METHOD PROTECTED DriveHomeAbsSwitch : BOOL
VAR_INPUT
	Execute: BOOL;
END_VAR

VAR_INST
	
	HomeSwState: INT; 
END_VAR
VAR
	
END_VAR


IF HomeRefTrig.EDGEPOS(Execute) THEN
	HomeSwState := 1;
	DriveHomeAbsSwitch := FALSE;
END_IF


IF HomeRefTrig.EDGENEG(Execute) THEN
	
	HomeSwState := 0;
END_IF



CASE HomeSwState OF
	0:
		DriveHomeAbsSwitch := FALSE;
	1:

		IF AxisCtrlPtr^.Input.Parameter.HomeOptions.stBasic.StartDirection = eHomeModeOption.ePOSITIVE THEN
		//Sensor positive
			IF AxisCtrlPtr^.Input.Parameter.HomeOptions.stAbsSwitch.SensorEdgeSignal = eHomeModeOption.ePOSITIVE THEN
				Homing_Ctrl_Params.HomingMethod := DINT_TO_SINT(eHomingMethods.HomeAbs);
			ELSE
				Homing_Ctrl_Params.HomingMethod := DINT_TO_SINT(eHomingMethods.ForwardOnNegSw);
			END_IF
		ELSE//Direction negative
			
			IF AxisCtrlPtr^.Input.Parameter.HomeOptions.stAbsSwitch.SensorEdgeSignal = eHomeModeOption.ePOSITIVE THEN
				Homing_Ctrl_Params.HomingMethod := DINT_TO_SINT(eHomingMethods.ReverseOnPosSw);
			ELSE
				Homing_Ctrl_Params.HomingMethod := DINT_TO_SINT(eHomingMethods.ReverseOnNegSw);
			END_IF
				
		END_IF
		

		HomeSwState := 2;
		Meth_Homing(FALSE);
	2:
		IF Meth_Homing(TRUE) THEN
		  Meth_Homing(FALSE);		  
		  HomeSwState := 3;
		END_IF
		
	3:
				//homin direct
		(*IF HomeDirect(TRUE) THEN*)   		 
			Meth_CoEChangOperationMode(FALSE,eCaOpDriveModeOfOperation.CyclicSyncMode);
			
			DriveHomeAbsSwitch := TRUE;
		//END_IF	
		
		
END_CASE
END_METHOD

METHOD DriveHomeLagError : BOOL
VAR_INPUT
	Execute: BOOL;
END_VAR

VAR_INST
//	State:INT;	
//	HomeTrig: Trigger;
//	Reset:BOOL;	
//	Delay:	TON;	
	HomeLagErrState: INT; 	
	LagErrorPrevState : INT;
	
END_VAR
VAR
	
END_VAR


IF HomeRefTrig.EDGEPOS(Execute) THEN
	HomeLagErrState := 1;
	DriveHomeLagError := FALSE;
END_IF


IF HomeRefTrig.EDGENEG(Execute) THEN
	
	HomeLagErrState := 0;
END_IF



CASE HomeLagErrState OF
	0:
	//
	
	//CoEDrive_Ctrl_Adr.MaxCurrent.Index
	1:
	// set min torque
		FB_EcCoeSdoWrite.bExecute := FALSE;
		
		HomeLagErrState := HomeLagErrState + 1;
	2:
		
			FB_EcCoeSdoWrite.sNetId		:= strEcNetId;
			FB_EcCoeSdoWrite.nSlaveAddr	:= io_EtherCatAddr;
			FB_EcCoeSdoWrite.nIndex		:= CoEDrive_Ctrl_Adr.MaxCurrent.Index; 
			FB_EcCoeSdoWrite.nSubIndex	:= CoEDrive_Ctrl_Adr.MaxCurrent.SunIndex; 
			FB_EcCoeSdoWrite.pSrcBuf	:= ADR(AxisCtrlPtr^.Input.Parameter.HomeOptions.stLagErr.BlockSearchMaxCurrent);
			FB_EcCoeSdoWrite.cbBufLen	:= SIZEOF(AxisCtrlPtr^.Input.Parameter.HomeOptions.stLagErr.BlockSearchMaxCurrent);
			FB_EcCoeSdoWrite.tTimeout	:= T#10S;
	
			FB_EcCoeSdoWrite.bExecute := TRUE;
			
			HomeLagErrState := HomeLagErrState + 1;
	3:
			
	
			IF NOT FB_EcCoeSdoWrite.bBusy THEN	
				IF NOT FB_EcCoeSdoWrite.bError THEN
					FB_EcCoeSdoWrite.bExecute		:= FALSE;
					HomeLagErrState :=  HomeLagErrState + 1;
				ELSE
					HomeLagErrState := 20;//error	
				END_IF	
			END_IF
			
	4:
		
			FB_EcCoeSdoWrite.sNetId		:= strEcNetId;
			FB_EcCoeSdoWrite.nSlaveAddr	:= io_EtherCatAddr;
			FB_EcCoeSdoWrite.nIndex		:= CoEDrive_Ctrl_Adr.MaxCurrent.Index; 
			FB_EcCoeSdoWrite.nSubIndex	:= CoEDrive_Ctrl_Adr.MaxCurrent.SunIndex; 
			FB_EcCoeSdoWrite.pSrcBuf	:= ADR(AxisCtrlPtr^.Input.Parameter.HomeOptions.stLagErr.BlockSearchRatedCurrent);
			FB_EcCoeSdoWrite.cbBufLen	:= SIZEOF(AxisCtrlPtr^.Input.Parameter.HomeOptions.stLagErr.BlockSearchRatedCurrent);
			FB_EcCoeSdoWrite.tTimeout	:= T#10S;
	
			FB_EcCoeSdoWrite.bExecute := TRUE;
			
			HomeLagErrState := HomeLagErrState + 1;
	5:
			
	
			IF NOT FB_EcCoeSdoWrite.bBusy THEN	
				IF NOT FB_EcCoeSdoWrite.bError THEN
					FB_EcCoeSdoWrite.bExecute		:= FALSE;
					HomeLagErrState :=  HomeLagErrState + 1;
				ELSE
					HomeLagErrState := 22;//error	
				END_IF	
			END_IF
			
			
	6:
		
			FB_EcCoeSdoWrite.sNetId		:= strEcNetId;
			FB_EcCoeSdoWrite.nSlaveAddr	:= io_EtherCatAddr;
			FB_EcCoeSdoWrite.nIndex		:= CoEDrive_Ctrl_Adr.PositionErrorWin.Index; 
			FB_EcCoeSdoWrite.nSubIndex	:= CoEDrive_Ctrl_Adr.PositionErrorWin.SunIndex; 
			FB_EcCoeSdoWrite.pSrcBuf	:= ADR(AxisCtrlPtr^.Input.Parameter.HomeOptions.stLagErr.BlockSearchPositionWindow);
			FB_EcCoeSdoWrite.cbBufLen	:= SIZEOF(AxisCtrlPtr^.Input.Parameter.HomeOptions.stLagErr.BlockSearchPositionWindow);
			FB_EcCoeSdoWrite.tTimeout	:= T#10S;
	
			FB_EcCoeSdoWrite.bExecute := TRUE;
			
			HomeLagErrState := HomeLagErrState + 1;
	7:
			
	
			IF NOT FB_EcCoeSdoWrite.bBusy THEN	
				IF NOT FB_EcCoeSdoWrite.bError THEN
					FB_EcCoeSdoWrite.bExecute		:= FALSE;
					HomeLagErrState :=  HomeLagErrState + 1;
				ELSE
					HomeLagErrState := 20;//error	
				END_IF	
			END_IF		
			
			
	8:	
		IF WriteNC_AxisBoolParam(MC_AxisParameter:=MC_AxisParameter.EnablePosLagMonitoring,ParamValue:=FALSE) THEN
				HomeLagErrState := HomeLagErrState + 1;
			END_IF		
		
	
	9:
	

		IF AxisCtrlPtr^.Input.Parameter.HomeOptions.stBasic.StartDirection = eHomeModeOption.ePOSITIVE THEN
		//Sensor positive
 				Homing_Ctrl_Params.HomingMethod := DINT_TO_SINT(eHomingMethods.HarsrStopPosDir);
			ELSE
				Homing_Ctrl_Params.HomingMethod := DINT_TO_SINT(eHomingMethods.HarsrStopNegDir);			
		END_IF
		

		HomeLagErrState :=  HomeLagErrState + 1;
		Meth_Homing(FALSE);
	10:
		IF Meth_Homing(TRUE) THEN
		  Meth_Homing(FALSE);		
 		  HomeLagErrState :=  HomeLagErrState + 1;
		  AxisCtrlPtr^.Input.Command.Power := FALSE;
		END_IF
	11:
			FB_EcCoeSdoWrite.sNetId		:= strEcNetId;
			FB_EcCoeSdoWrite.nSlaveAddr	:= io_EtherCatAddr;
			FB_EcCoeSdoWrite.nIndex		:= CoEDrive_Ctrl_Adr.MaxCurrent.Index; 
			FB_EcCoeSdoWrite.nSubIndex	:= CoEDrive_Ctrl_Adr.MaxCurrent.SunIndex; 
			FB_EcCoeSdoWrite.pSrcBuf	:= ADR(AxisCtrlPtr^.Input.Parameter.HomeOptions.stLagErr.BlockSearchMaxCurrent);
			FB_EcCoeSdoWrite.cbBufLen	:= SIZEOF(AxisCtrlPtr^.Input.Parameter.HomeOptions.stLagErr.BlockSearchMaxCurrent);
			FB_EcCoeSdoWrite.tTimeout	:= T#10S;
	
			FB_EcCoeSdoWrite.bExecute := TRUE;
			
			HomeLagErrState := HomeLagErrState + 1;	
		
	12:
			IF NOT FB_EcCoeSdoWrite.bBusy THEN	
				IF NOT FB_EcCoeSdoWrite.bError THEN
					FB_EcCoeSdoWrite.bExecute		:= FALSE;
					HomeLagErrState :=  HomeLagErrState + 1;
				ELSE
					HomeLagErrState := 20;//error	
				END_IF	
			END_IF	
			
	13:
			FB_EcCoeSdoWrite.sNetId		:= strEcNetId;
			FB_EcCoeSdoWrite.nSlaveAddr	:= io_EtherCatAddr;
			FB_EcCoeSdoWrite.nIndex		:= CoEDrive_Ctrl_Adr.PositionErrorWin.Index; 
			FB_EcCoeSdoWrite.nSubIndex	:= CoEDrive_Ctrl_Adr.PositionErrorWin.SunIndex; 
			FB_EcCoeSdoWrite.pSrcBuf	:= ADR(AxisCtrlPtr^.Input.Parameter.HomeOptions.stLagErr.BlockExitPositionWindow);
			FB_EcCoeSdoWrite.cbBufLen	:= SIZEOF(AxisCtrlPtr^.Input.Parameter.HomeOptions.stLagErr.BlockExitPositionWindow);;
			FB_EcCoeSdoWrite.tTimeout	:= T#10S;
	
			FB_EcCoeSdoWrite.bExecute := TRUE;
			
			HomeLagErrState := HomeLagErrState + 1;	
		
	14:
			IF NOT FB_EcCoeSdoWrite.bBusy THEN	
				IF NOT FB_EcCoeSdoWrite.bError THEN
					FB_EcCoeSdoWrite.bExecute		:= FALSE;
					HomeLagErrState :=  HomeLagErrState + 1;
				ELSE
					HomeLagErrState := 20;//error	
				END_IF	
			END_IF	

	15:
		
			FB_EcCoeSdoWrite.sNetId		:= strEcNetId;
			FB_EcCoeSdoWrite.nSlaveAddr	:= io_EtherCatAddr;
			FB_EcCoeSdoWrite.nIndex		:= CoEDrive_Ctrl_Adr.MaxCurrent.Index; 
			FB_EcCoeSdoWrite.nSubIndex	:= CoEDrive_Ctrl_Adr.MaxCurrent.SunIndex; 
			FB_EcCoeSdoWrite.pSrcBuf	:= ADR(AxisCtrlPtr^.Input.Parameter.HomeOptions.stLagErr.BlockExitRatedCurrent);
			FB_EcCoeSdoWrite.cbBufLen	:= SIZEOF(AxisCtrlPtr^.Input.Parameter.HomeOptions.stLagErr.BlockExitRatedCurrent);
			FB_EcCoeSdoWrite.tTimeout	:= T#10S;
	
			FB_EcCoeSdoWrite.bExecute := TRUE;
			
			HomeLagErrState := HomeLagErrState + 1;
	16:
			
	
			IF NOT FB_EcCoeSdoWrite.bBusy THEN	
				IF NOT FB_EcCoeSdoWrite.bError THEN
					FB_EcCoeSdoWrite.bExecute		:= FALSE;
					HomeLagErrState :=  HomeLagErrState + 1;
				ELSE
					HomeLagErrState := 22;//error	
				END_IF	
			END_IF

		
	17:	
 		AxisCtrlPtr^.Input.Command.Power := TRUE;
		DriveHomeLagError:= TRUE;
	
		
END_CASE

	IF LagErrorPrevState <> HomeLagErrState THEN
		fnLogMsg(ADR(LogMsg_0),LOG_INFO,'Coe Basic Drive Lag Err step %d',HomeLagErrState,0,0);
		LagErrorPrevState := HomeLagErrState;
	END_IF
END_METHOD

METHOD PROTECTED DriveHomeRefPulse : BOOL
VAR_INPUT
	Execute: BOOL;
END_VAR

VAR_INST
	 
	RefState: INT; 
	PrevRefState : INT;
END_VAR
VAR
	
END_VAR


IF HomeRefTrig.EDGEPOS(Execute) THEN
	RefState := 1;
	DriveHomeRefPulse := FALSE;
END_IF


IF HomeRefTrig.EDGENEG(Execute) THEN
	
	RefState := 0;
END_IF



CASE RefState OF
	0:
		DriveHomeRefPulse := FALSE;
	1:
 
		IF AxisCtrlPtr^.Input.Parameter.HomeOptions.stBasic.StartDirection = eHomeModeOption.ePOSITIVE THEN
			Homing_Ctrl_Params.HomingMethod := DINT_TO_SINT(eHomingMethods.IndexPulsePosDir);
		ELSE
			Homing_Ctrl_Params.HomingMethod := DINT_TO_SINT(eHomingMethods.IndexPulseNegDir);
		END_IF	
		RefState := RefState  +1 ;
		Meth_Homing(FALSE);
	2:
		IF Meth_Homing(TRUE) THEN
		  Meth_Homing(FALSE);
		  RefState := RefState  +1 ;
		  DriveHomeRefPulse := TRUE;
		END_IF
	3:
				//homin direct
	//	IF HomeDirect(TRUE) THEN   		 
			Meth_CoEChangOperationMode(FALSE,eCaOpDriveModeOfOperation.CyclicSyncMode);
			RefState := RefState  +1 ;
	//	END_IF
	
	4: 	
	   	  DriveHomeRefPulse := TRUE;
		
		
		
END_CASE


	IF PrevRefState <> RefState THEN
		fnLogMsg(ADR(LogMsg_0),LOG_INFO,'Coe Basic Home Ref Pulse step %d',RefState,0,0);
		PrevRefState := RefState;
	END_IF
END_METHOD

METHOD DriveUnitsTorqueToRealValue : LREAL
VAR_INPUT
	
	Torque: LREAL;	

END_VAR
DriveUnitsTorqueToRealValue := Torque;
END_METHOD

METHOD EcCoeSdoRead : BOOL
VAR_INPUT
	Execute: 	BOOL;
END_VAR

VAR_INST
	CoReaderrorTrig: 		Trigger ;	
	
END_VAR

IF CoReaderrorTrig.EDGEPOS(Execute) THEN
	EcCoeSdoRead:= FALSE;
	StateCoeSdoRead	:= 1;		
END_IF

IF CoReaderrorTrig.EDGENEG(Execute) THEN
	
	CoeSdoRW.Output.Read.Done 	:= FALSE;
	FB_EcCoeSdoRead_0.bExecute 	:= FALSE;
	StateCoeSdoRead		:= 0;	
	EcCoeSdoRead		:= FALSE;
	
END_IF


CASE StateCoeSdoRead OF
	
	0:
		// Wait	
	1:
		FB_EcCoeSdoRead_0.sNetId		:= F_CreateAmsNetId(AxisCtrlPtr^.Input.Parameter.ecNetIdArr); 
		FB_EcCoeSdoRead_0.nSlaveAddr	:= io_EtherCatAddr;
		FB_EcCoeSdoRead_0.nSubIndex		:= CoeSdoRW.Input.Read.nSubIndex;
		FB_EcCoeSdoRead_0.nIndex		:= CoeSdoRW.Input.Read.nIndex; 
		FB_EcCoeSdoRead_0.pDstBuf		:= CoeSdoRW.Input.Read.pDstBuf; 
		FB_EcCoeSdoRead_0.cbBufLen		:= CoeSdoRW.Input.Read.cbBufLen; 
		FB_EcCoeSdoRead_0.tTimeout		:= CoeSdoRW.Input.Read.tTimeout; 
		StateCoeSdoRead	:= 2;
		FB_EcCoeSdoRead_0.bExecute		:= FALSE;
		
	2:	

		FB_EcCoeSdoRead_0.bExecute		:= TRUE;	
		IF (FB_EcCoeSdoRead_0.bBusy = TRUE) THEN
			StateCoeSdoRead	:= 3;	
		END_IF

	3:	
		IF (FB_EcCoeSdoRead_0.bBusy = FALSE) THEN
			
			CoeSdoRW.Output.Read.Done	:= TRUE;
			EcCoeSdoRead	:= TRUE;
			StateCoeSdoRead	:= 4;	
		END_IF
	
	4:	
		FB_EcCoeSdoRead_0.bExecute	:= FALSE;
		EcCoeSdoRead	:= TRUE;
	
		
END_CASE

FB_EcCoeSdoRead_0();

(* check if error occured *)
IF errorTrig.EDGEPOS(FB_EcCoeSdoRead_0.bError) THEN
	
	// Add FB Error to ErrorHandler	
	AddNCError(FB_EcCoeSdoRead_0.nErrId,'NC Error FB_EcCoeSdoRead_0 ErrorID: ');
	
	EcCoeSdoRead :=  FALSE ;
	FB_EcCoeSdoRead_0.bExecute := FALSE;
END_IF

CoeSdoRW.Output.Read.Busy	:= FB_EcCoeSdoRead_0.bBusy;
END_METHOD

METHOD EcCoeSdoWrite : BOOL
VAR_INPUT
	Execute: 	BOOL;
END_VAR

VAR_INST
	CanOpWriteErrorTrig: 		Trigger ;	
	
END_VAR
VAR_OUTPUT	
	Error: 	BOOL;
END_VAR

IF CanOpWriteErrorTrig.EDGEPOS(Execute) THEN
	EcCoeSdoWrite		:= FALSE;
	StateCoeSdoWrite	:= 1;		
	Error 				:= FALSE;
END_IF

IF CanOpWriteErrorTrig.EDGENEG(Execute) THEN
	
	CoeSdoRW.Output.Write.Done 	:= FALSE;
	FB_EcCoeSdoWrite_0.bExecute := FALSE;
	StateCoeSdoWrite	:= 0;	
	EcCoeSdoWrite		:= FALSE;
	
END_IF


CASE StateCoeSdoWrite OF
	
	0:
		// Wait	
	1:										   
		FB_EcCoeSdoWrite_0.sNetId		:= F_CreateAmsNetId(AxisCtrlPtr^.Input.Parameter.ecNetIdArr); 
		FB_EcCoeSdoWrite_0.nSlaveAddr	:= AxisCtrlPtr^.Input.Parameter.Drive.EtherCatAddr;
		FB_EcCoeSdoWrite_0.nSubIndex	:= CoeSdoRW.Input.Write.nSubIndex;
		FB_EcCoeSdoWrite_0.nIndex		:= CoeSdoRW.Input.Write.nIndex; 
		FB_EcCoeSdoWrite_0.pSrcBuf		:= CoeSdoRW.Input.Write.pSrcBuf; 
		FB_EcCoeSdoWrite_0.cbBufLen		:= CoeSdoRW.Input.Write.cbBufLen; 
		FB_EcCoeSdoWrite_0.tTimeout		:= CoeSdoRW.Input.Write.tTimeout; 
		StateCoeSdoWrite	:= 2;	
	2:	

		FB_EcCoeSdoWrite_0.bExecute		:= TRUE;	
		IF (FB_EcCoeSdoWrite_0.bBusy = TRUE) THEN
			StateCoeSdoWrite	:= 3;	
		END_IF

	3:	
		IF (FB_EcCoeSdoWrite_0.bBusy = FALSE) THEN
			FB_EcCoeSdoWrite_0.bExecute		:= FALSE;
			CoeSdoRW.Output.Write.Done		:= TRUE;
			EcCoeSdoWrite		:= TRUE;
			StateCoeSdoWrite	:= 4;	
		ELSIF FB_EcCoeSdoWrite_0.bError THEN
			Error := TRUE;
		END_IF
	4:
		EcCoeSdoWrite		:= TRUE;
	
	
END_CASE

FB_EcCoeSdoWrite_0();

(* check if error occured *)
IF errorTrig.EDGEPOS(FB_EcCoeSdoWrite_0.bError) THEN
	
	// Add FB Error to ErrorHandler	
	AddNCError(FB_EcCoeSdoWrite_0.nErrId,'NC Error FB_EcCoeSdoWrite_0 ErrorID: ');
	
	EcCoeSdoWrite :=  FALSE ;
	FB_EcCoeSdoWrite_0.bExecute := FALSE;
END_IF

CoeSdoRW.Output.Write.Busy	:= FB_EcCoeSdoWrite_0.bBusy;
END_METHOD

METHOD GetCanOpenAdr : BOOL
VAR_INPUT
END_VAR


VAR
	
	SpeedSwSubIndex: INT;
END_VAR
	
	CoEDrive_Ctrl_Adr.OperationMode.Index 	   := 16#6060;
	CoEDrive_Ctrl_Adr.OperationMode.SunIndex   := 0;
	CoEDrive_Ctrl_Adr.OperationMode.Size	   := 1;

	CoEDrive_Ctrl_Adr.ControlWord.Index   	 := 16#6040;	
	CoEDrive_Ctrl_Adr.ControlWord.SunIndex   := 0;
	CoEDrive_Ctrl_Adr.ControlWord.Size       := 2;
	
	
	CoEDrive_Ctrl_Adr.HomingMethod.Index  := 16#6098;
	CoEDrive_Ctrl_Adr.HomingMethod.SunIndex  := 0;
	CoEDrive_Ctrl_Adr.HomingMethod.Size      := 1;
	
	
	CoEDrive_Ctrl_Adr.HomingSWSpeed.Index     := 16#6099;		
	CoEDrive_Ctrl_Adr.HomingSWSpeed.SunIndex  := 1;
	CoEDrive_Ctrl_Adr.HomingSWSpeed.Size      := 4;
	
	
	CoEDrive_Ctrl_Adr.HomingTrSpeed.Index    := 16#6099;
	CoEDrive_Ctrl_Adr.HomingTrSpeed.SunIndex := 2;
	CoEDrive_Ctrl_Adr.HomingTrSpeed.Size     := 4;
	
	
	
	CoEDrive_Ctrl_Adr.HomingAcc.Index     	 := 16#609A;
	CoEDrive_Ctrl_Adr.HomingAcc.SunIndex  	 := 0;
	CoEDrive_Ctrl_Adr.HomingAcc.Size      := 4;
	
	CoEDrive_Ctrl_Adr.HomeOffset.Index    	 := 16#607C;
	CoEDrive_Ctrl_Adr.HomeOffset.SunIndex  	 := 0;
	CoEDrive_Ctrl_Adr.HomeOffset.Size      := 4;

	
	CoEDrive_Ctrl_Adr.StatusWord.Index     := 16#6041;
	CoEDrive_Ctrl_Adr.StatusWord.SunIndex  := 0;
	CoEDrive_Ctrl_Adr.StatusWord.Size      := 2;
	
	CoEDrive_Ctrl_Adr.PositionErrorWin.Index 	:= 16#6065;
	CoEDrive_Ctrl_Adr.PositionErrorWin.SunIndex := 	0;	
	CoEDrive_Ctrl_Adr.PositionErrorWin.Size 	:= 4;     
	
	
	CoEDrive_Ctrl_Adr.MaxTorque.Index 	  := 16#6072;
	CoEDrive_Ctrl_Adr.MaxTorque.SunIndex  := 0;
	CoEDrive_Ctrl_Adr.MaxTorque.Size      := 2;
	
	CoEDrive_Ctrl_Adr.MaxCurrent.Index 	  := 16#6073;
	CoEDrive_Ctrl_Adr.MaxCurrent.SunIndex  := 0;
	CoEDrive_Ctrl_Adr.MaxCurrent.Size      := 2;
	
	CoEDrive_Ctrl_Adr.RatedCurrent.Index     := 16#6075;
	CoEDrive_Ctrl_Adr.RatedCurrent.SunIndex  := 0;
	CoEDrive_Ctrl_Adr.RatedCurrent.Size      := 4;
	
 
	
	

	
	CoEDrive_Ctrl_Adr.TorqueOffset.Index 	 := 16#60B2; // integer 16
	CoEDrive_Ctrl_Adr.TorqueOffset.SunIndex  := 0;
	CoEDrive_Ctrl_Adr.TorqueOffset.Size      := 2;


	
	
    //VeloctyCtrlTN
END_METHOD

METHOD GetErrCanAdr : BOOL
VAR_INPUT
END_VAR


VAR
	
END_VAR
CoeErrIdIndex	:= 16#603F;
END_METHOD

METHOD IsHomingAttained : BOOL
VAR_INPUT
END_VAR
	

IF io_StatusWord.12 <>0 THEN
	IsHomingAttained :=TRUE;
ELSE
	IsHomingAttained :=FALSE;
END_IF
END_METHOD

METHOD Meth_ChangingOperationMode : BOOL
VAR_INPUT
	Execute   : BOOL;
	OperMode : eDriveModeOfOperation; 
	
END_VAR
VAR_INST
	
	CngOperState : INT;
	Mode      : USINT;	
END_VAR

VAR
	
	ChangeDone : BOOL;
END_VAR
IF ChangeModeOperTrig.EDGEPOS(Execute) THEN

	Meth_ChangingOperationMode := FALSE;				
	Mode := DINT_TO_USINT(OperMode);
	ChangeDone := FALSE;
	CngOperState := 1;

	
END_IF


IF ChangeModeOperTrig.EDGENEG(Execute) THEN
	
	CngOperState := 0;
END_IF



CASE CngOperState OF
	0:
		Meth_CoEChangOperationMode(FALSE,eCaOpDriveModeOfOperation.ProfilePositionMode);
		
	1: 
		//Meth_CoEChangOperationMode
		CASE OperMode OF
			eDriveModeOfOperation.ProfilePositionMode				:
				IF Meth_CoEChangOperationMode(TRUE,eCaOpDriveModeOfOperation.ProfilePositionMode) THEN
					ChangeDone := TRUE;
				END_IF
				
		    eDriveModeOfOperation.VelocityCtrMode    				:
				IF Meth_CoEChangOperationMode(TRUE,eCaOpDriveModeOfOperation.VelocityCtrMode)THEN
					ChangeDone := TRUE;
				END_IF
		    eDriveModeOfOperation.ProfileVelocityMode 	   	    :
				IF Meth_CoEChangOperationMode(TRUE,eCaOpDriveModeOfOperation.ProfileVelocityMode) THEN
					ChangeDone := TRUE;
				END_IF
				
		    eDriveModeOfOperation.TorqueVelocityMode 				:
				IF Meth_CoEChangOperationMode(TRUE,eCaOpDriveModeOfOperation.TorqueVelocityMode) THEN
					ChangeDone := TRUE;
				END_IF
				
		    eDriveModeOfOperation.HomingMode				    	:
				IF Meth_CoEChangOperationMode(TRUE,eCaOpDriveModeOfOperation.HomingMode)THEN
					ChangeDone := TRUE;
				END_IF
				
		    eDriveModeOfOperation.InterpolationPosMode			:
				IF Meth_CoEChangOperationMode(TRUE,eCaOpDriveModeOfOperation.InterpolationPosMode) THEN
					ChangeDone := TRUE;
				END_IF
		    eDriveModeOfOperation.CyclicSyncMode					:
				Meth_CoEChangOperationMode(TRUE,eCaOpDriveModeOfOperation.CyclicSyncMode);
		END_CASE
		CngOperState := 2;

	2:
 		Meth_ChangingOperationMode := TRUE;
		
		
END_CASE
END_METHOD

METHOD Meth_CngMaxTorque : BOOL
VAR_INPUT
	Execute   : BOOL;
	Value	  : LREAL;
END_VAR


VAR


	
END_VAR
VAR_INST
	//
	CngMaxTorqueTrigger : Trigger ;
	CngMaxTorqueState   : SINT;	
	
END_VAR


VAR_OUTPUT
	Error : BOOL;
END_VAR

IF CngMaxTorqueTrigger.EDGEPOS(Execute) THEN
	Meth_CngMaxTorque := FALSE;
	CngMaxTorqueState := 1;
END_IF


IF CngMaxTorqueTrigger.EDGENEG(Execute) THEN
	CngMaxTorqueState := 0;
	Meth_CngMaxTorque := FALSE;
	EcCoeSdoWrite(FALSE);

END_IF

IF NOT AxisCtrlPtr^.Output.Status.Drive.ActiveHW THEN// SIM
	Meth_CngMaxTorque := TRUE;
ELSE


CASE CngMaxTorqueState OF 
	0:
	
		Meth_CngMaxTorque := FALSE;
	1:
		
		CoeSdoRW.Input.Write.nIndex    := CoEDrive_Ctrl_Adr.MaxTorque.Index;	  
		CoeSdoRW.Input.Write.nSubIndex := CoEDrive_Ctrl_Adr.MaxTorque.SunIndex;
		UintValue := LREAL_TO_UINT(Meth_TorqueInDriveUnits( Value));
		CoeSdoRW.Input.Write.pSrcBuf   :=   ADR(UintValue); 	 
		CoeSdoRW.Input.Write.cbBufLen  := SIZEOF(UintValue)  ; 
		 
		IF EcCoeSdoWrite(TRUE , Error=> Error ) THEN
			
			CngMaxTorqueState := CngMaxTorqueState +1;
		END_IF
	
	2:
		Meth_CngMaxTorque := TRUE;

END_CASE

END_IF
END_METHOD

METHOD Meth_CngTorqueOffset : BOOL
VAR_INPUT
	Execute   : BOOL;
	Value	  : LREAL;
END_VAR

VAR_INST
		//
	CngTorqueOffsetTrigger : Trigger ;
	CngTorqueOffsetState   : SINT;	
	
END_VAR
 
VAR_OUTPUT
	Error : BOOL;
END_VAR

IF CngTorqueOffsetTrigger.EDGEPOS(Execute) THEN
	Meth_CngTorqueOffset := FALSE;
	CngTorqueOffsetState := 1;	
END_IF


IF CngTorqueOffsetTrigger.EDGENEG(Execute) THEN
	CngTorqueOffsetState := 0;
	Meth_CngTorqueOffset := FALSE;
	EcCoeSdoWrite(FALSE);

END_IF
IF NOT AxisCtrlPtr^.Output.Status.Drive.ActiveHW THEN// SIM
	Meth_CngTorqueOffset := TRUE;
ELSE


CASE CngTorqueOffsetState OF 
	0:
		Meth_CngTorqueOffset := FALSE;
	1:
		
		CoeSdoRW.Input.Write.nIndex    := CoEDrive_Ctrl_Adr.TorqueOffset.Index ;		
		CoeSdoRW.Input.Write.nSubIndex := CoEDrive_Ctrl_Adr.TorqueOffset.SunIndex; 	
	    CoeSdoRW.Input.Write.cbBufLen  := CoEDrive_Ctrl_Adr.TorqueOffset.Size;     	
		UintValue := LREAL_TO_UINT(Meth_TorqueInDriveUnits( Value));
		CoeSdoRW.Input.Write.pSrcBuf   :=   ADR(UintValue); 	 	 
		 
		IF EcCoeSdoWrite(TRUE , Error=> Error ) THEN
			fnLogMsg(ADR(LogMsg_0),LOG_INFO,'Meth Change torque Offset %d After convert',UintValue,0,0);
			CngTorqueOffsetState := CngTorqueOffsetState +1;
		END_IF
	
	2:
		Meth_CngTorqueOffset := TRUE;

END_CASE

END_IF
END_METHOD

METHOD Meth_CoEChangOperationMode : BOOL
VAR_INPUT
	Execute   : BOOL;	
	OperMode :eCaOpDriveModeOfOperation; 
END_VAR
VAR_INST
	ConfigHomeTrig  : 	Trigger;
	CngOperState : INT;
	Mode      : USINT;	
END_VAR

VAR
	
	
END_VAR
IF ConfigHomeTrig.EDGEPOS(Execute) THEN

	Meth_CoEChangOperationMode := FALSE;				
	Mode := DINT_TO_USINT(OperMode);

	CngOperState := 1;
END_IF


IF ConfigHomeTrig.EDGENEG(Execute) THEN
	
	CngOperState := 0;
END_IF



CASE CngOperState OF
	0:
		FB_EcCoeSdoWrite.bExecute := FALSE;
		Meth_CoEChangOperationMode := 0;
	1: 
		IF NOT FB_EcCoeSdoWrite.bBusy THEN	
			//Config homing mehod
			FB_EcCoeSdoWrite.sNetId		:= strEcNetId;
			FB_EcCoeSdoWrite.nSlaveAddr	:= io_EtherCatAddr;
			FB_EcCoeSdoWrite.nIndex		:= CoEDrive_Ctrl_Adr.OperationMode.Index; 
			FB_EcCoeSdoWrite.nSubIndex	:= CoEDrive_Ctrl_Adr.OperationMode.SunIndex; 
			FB_EcCoeSdoWrite.pSrcBuf	:= ADR(Mode);
			FB_EcCoeSdoWrite.cbBufLen	:= SIZEOF(Mode);
			FB_EcCoeSdoWrite.tTimeout	:= T#10S;
			
			FB_EcCoeSdoWrite.bExecute		:= TRUE;
		END_IF
		CngOperState := 2;

	2:
		IF NOT FB_EcCoeSdoWrite.bBusy THEN	
			IF NOT FB_EcCoeSdoWrite.bError THEN
				FB_EcCoeSdoWrite.bExecute		:= FALSE;				
				Meth_CoEChangOperationMode := TRUE;
			ELSE
				fnLogMsg(ADR(LogMsg_0),LOG_ERROR,'NO LINKS FOR DRIVE',0,0,0);	
				Meth_CoEChangOperationMode := FALSE;		
			END_IF	
			
		END_IF	
		
		
END_CASE
END_METHOD

METHOD Meth_ConfigHomeParamters : BOOL
VAR_INPUT
	Execute   : BOOL;	
END_VAR
VAR_INST
	ConfigHomeTrig  : 	Trigger;
	ConfigHomeState : INT;
END_VAR
IF ConfigHomeTrig.EDGEPOS(Execute) THEN

	Meth_ConfigHomeParamters := FALSE;				


	ConfigHomeState := 1;
END_IF


IF ConfigHomeTrig.EDGENEG(Execute) THEN
	
	ConfigHomeState := 0;
END_IF


CASE ConfigHomeState OF
	0:
		FB_EcCoeSdoWrite.bExecute := FALSE;
	1: 
			
		//Config homing mehod
		FB_EcCoeSdoWrite.sNetId			:= strEcNetId;
		FB_EcCoeSdoWrite.nSlaveAddr		:= WORD_TO_UINT(io_EtherCatAddr);
		FB_EcCoeSdoWrite.nIndex			:= CoEDrive_Ctrl_Adr.HomingMethod.Index; 
		FB_EcCoeSdoWrite.nSubIndex		:= CoEDrive_Ctrl_Adr.HomingMethod.SunIndex; 
		FB_EcCoeSdoWrite.pSrcBuf		:= ADR(Homing_Ctrl_Params.HomingMethod);
		FB_EcCoeSdoWrite.cbBufLen		:= SIZEOF(Homing_Ctrl_Params.HomingMethod);
		FB_EcCoeSdoWrite.tTimeout		:= T#10S;
		
		FB_EcCoeSdoWrite.bExecute		:= TRUE;
		
		ConfigHomeState := 12;
		
		NextState := 2;
	2: //Config Homing SW Speed
	
		FB_EcCoeSdoWrite.sNetId		:= strEcNetId;
		FB_EcCoeSdoWrite.nSlaveAddr	:= WORD_TO_UINT(io_EtherCatAddr);
		FB_EcCoeSdoWrite.nIndex		:= CoEDrive_Ctrl_Adr.HomingSWSpeed.Index; 
		FB_EcCoeSdoWrite.nSubIndex	:= CoEDrive_Ctrl_Adr.HomingSWSpeed.SunIndex; 
		FB_EcCoeSdoWrite.pSrcBuf	:= ADR(Homing_Ctrl_Params.HomingSWSpeed);
		FB_EcCoeSdoWrite.cbBufLen	:= SIZEOF(Homing_Ctrl_Params.HomingSWSpeed);
		FB_EcCoeSdoWrite.tTimeout	:= T#10S;
		
		FB_EcCoeSdoWrite.bExecute		:= TRUE;
		
		ConfigHomeState := 12;
		
		NextState := 3;
	3: //Config Homing Trigger Speed
		FB_EcCoeSdoWrite.sNetId		:= strEcNetId;
		FB_EcCoeSdoWrite.nSlaveAddr	:= WORD_TO_UINT(io_EtherCatAddr);
		FB_EcCoeSdoWrite.nIndex		:= CoEDrive_Ctrl_Adr.HomingTrSpeed.Index; 
		FB_EcCoeSdoWrite.nSubIndex	:= CoEDrive_Ctrl_Adr.HomingTrSpeed.SunIndex; 
		FB_EcCoeSdoWrite.pSrcBuf	:= ADR(Homing_Ctrl_Params.HomingTrSpeed);
		FB_EcCoeSdoWrite.cbBufLen	:= SIZEOF(Homing_Ctrl_Params.HomingTrSpeed);
		FB_EcCoeSdoWrite.tTimeout	:= T#10S;
		
		FB_EcCoeSdoWrite.bExecute		:= TRUE;


		
		ConfigHomeState := 12;
		
		NextState := 4;
		
	4:	//Config Homing SW Acc
	
		FB_EcCoeSdoWrite.sNetId		:= strEcNetId;
		FB_EcCoeSdoWrite.nSlaveAddr	:= WORD_TO_UINT(io_EtherCatAddr);
		FB_EcCoeSdoWrite.nIndex		:= CoEDrive_Ctrl_Adr.HomingAcc.Index; 
		FB_EcCoeSdoWrite.nSubIndex	:= CoEDrive_Ctrl_Adr.HomingAcc.SunIndex; 
		FB_EcCoeSdoWrite.pSrcBuf	:= ADR(Homing_Ctrl_Params.HomingAcc);
		FB_EcCoeSdoWrite.cbBufLen	:= SIZEOF(Homing_Ctrl_Params.HomingAcc);
		FB_EcCoeSdoWrite.tTimeout	:= T#10S;
		
		FB_EcCoeSdoWrite.bExecute		:= TRUE;
		ConfigHomeState := 12;
		
		NextState := 5;
	5://Config Offset
		FB_EcCoeSdoWrite.sNetId		:= strEcNetId;
		FB_EcCoeSdoWrite.nSlaveAddr	:=  WORD_TO_UINT(io_EtherCatAddr);
		FB_EcCoeSdoWrite.nIndex		:= CoEDrive_Ctrl_Adr.HomeOffset.Index; 
		FB_EcCoeSdoWrite.nSubIndex	:= CoEDrive_Ctrl_Adr.HomeOffset.SunIndex; 
		FB_EcCoeSdoWrite.pSrcBuf		:= ADR(Homing_Ctrl_Params.HomingOffset);
		FB_EcCoeSdoWrite.cbBufLen		:= SIZEOF(Homing_Ctrl_Params.HomingOffset);
		FB_EcCoeSdoWrite.tTimeout		:= T#10S;
		
		FB_EcCoeSdoWrite.bExecute		:= TRUE;

	
		ConfigHomeState := 12;
		
		NextState := 6;

	6://Done
		Meth_ConfigHomeParamters := TRUE;
	12:
		IF NOT FB_EcCoeSdoWrite.bBusy THEN	
			IF NOT FB_EcCoeSdoWrite.bError THEN
				FB_EcCoeSdoWrite.bExecute		:= FALSE;
				ConfigHomeState := NextState;
			ELSE
				NextState := 20;//error	
			END_IF	
			
		END_IF	
		
		
END_CASE
END_METHOD

METHOD Meth_DriveFWUpdate : BOOL
VAR_INPUT
	Execute:		BOOL;
END_VAR
VAR_INST
	UpdateDriveParamsTrig  : 	Trigger;
	UpdateFWState : INT;
	
	 
END_VAR
IF UpdateDriveParamsTrig.EDGEPOS(Execute) THEN
	
	UpdateFWState := 0;
	AxisCtrlPtr^.Output.Status.Drive.eUpdate_Staus := enum_DriveUpdateStatus.NoAction;
	AxisCtrlPtr^.Output.monitor.FileUpdate.FileUpdate_Error   := 	enum_DriveUpdateError.NoError;
	AxisCtrlPtr^.Output.monitor.FileUpdate.ErrorID := 0;
END_IF



CASE UpdateFWState OF 
	0://init -wait	

		
		UpdateFWState:=UpdateFWState +1;
	
	1://read Version Drive Param Version	
		// := 'Read Version';			
							
		CoeSdoRW.Input.Read.nIndex 	  := CoEDrive_Ctrl_Adr.FWVersionObj.Index; 
		CoeSdoRW.Input.Read.nSubIndex := CoEDrive_Ctrl_Adr.FWVersionObj.SunIndex;
		CoeSdoRW.Input.Read.pDstBuf	  := ADR(FOE_Ctrl_UpdateFW.Version_From_Drive);
 		CoeSdoRW.Input.Read.cbBufLen  := SIZEOF(FOE_Ctrl_UpdateFW.Version_From_Drive);  

		FOE_Ctrl_UpdateFW.fbFileOpen.bExecute    := FALSE;
		FOE_Ctrl_UpdateFW.fbFileClose.bExecute   := FALSE;
		FOE_Ctrl_UpdateFW.fbEcFoeLoad_0.bExecute := FALSE;
		EcCoeSdoRead(FALSE);
		FOE_Ctrl_UpdateFW.Foe_File_Path:=	AxisCtrlPtr^.Input.Parameter.Drive.sFoeFWFile_Path;
		UpdateFWState:= UpdateFWState +1;

		
	2://Download to Drive 
		// := 'Download to Drive';
		IF EcCoeSdoRead(TRUE) THEN		
  				
			AxisCtrlPtr^.Output.Status.Drive.ParamVer:=	FOE_Ctrl_UpdateFW.Version_From_Drive;	
			IF AxisCtrlPtr^.Output.Status.Drive.ParamVer <> AxisCtrlPtr^.Input.Parameter.Drive.LatestParamVer THEN				
				AxisCtrlPtr^.Output.Status.Drive.eUpdate_Staus:= enum_DriveUpdateStatus.Checking;
				UpdateFWState:=UpdateFWState +1;
			ELSE
				AxisCtrlPtr^.Output.Status.Drive.eUpdate_Staus:= enum_DriveUpdateStatus.Updated;
				UpdateFWState:=	100;										
			END_IF
						
		END_IF
		
	3: 
		
						
		FOE_Ctrl_UpdateFW.fbFileOpen.sNetId		:= ''; 
		FOE_Ctrl_UpdateFW.fbFileOpen.sPathName		:=FOE_Ctrl_UpdateFW.Foe_File_Path; 
		FOE_Ctrl_UpdateFW.fbFileOpen.nMode			:=FOPEN_MODEREAD; 
		FOE_Ctrl_UpdateFW.fbFileOpen.ePath			:=PATH_GENERIC ;
		
		FOE_Ctrl_UpdateFW.fbFileOpen.bExecute:=	TRUE; 

		UpdateFWState:=UpdateFWState +1;
	4:
		//Check Valid file Path
		// := 'Cheack Valid Path';
		
		IF FOE_Ctrl_UpdateFW.fbFileOpen.bBusy =FALSE AND FOE_Ctrl_UpdateFW.fbFileOpen.bError =FALSE THEN 
			FOE_Ctrl_UpdateFW.hFile := FOE_Ctrl_UpdateFW.fbFileOpen.hFile;
			FOE_Ctrl_UpdateFW.fbFileOpen.bExecute:=	FALSE;
			UpdateFWState:=UpdateFWState +1;
			
			
			
			
		ELSIF FOE_Ctrl_UpdateFW.fbFileOpen.bError =TRUE THEN 
			AxisCtrlPtr^.Output.Status.Drive.eUpdate_Staus 			  :=	enum_DriveUpdateStatus.Error;
			AxisCtrlPtr^.Output.monitor.FileUpdate.FileUpdate_Error   := 	enum_DriveUpdateError.FileNotFound;
			AxisCtrlPtr^.Output.monitor.FileUpdate.ErrorID 			  :=    FOE_Ctrl_UpdateFW.fbFileOpen.nErrId;
			UpdateFWState:=	11;				
		END_IF	
	5:
			FOE_Ctrl_UpdateFW.fbFileClose.bExecute:=	TRUE;	
			UpdateFWState:=UpdateFWState +1;
	6:	
		// := 'Close path';
		
		IF FOE_Ctrl_UpdateFW.fbFileClose.bBusy =FALSE AND FOE_Ctrl_UpdateFW.fbFileClose.bError =FALSE THEN 
			FOE_Ctrl_UpdateFW.fbFileClose.bExecute:=FALSE;	
			UpdateFWState:=UpdateFWState +1;

			
	
		ELSIF FOE_Ctrl_UpdateFW.fbFileClose.bError =TRUE THEN 
			AxisCtrlPtr^.Output.Status.Drive.eUpdate_Staus :=	enum_DriveUpdateStatus.Error;
			AxisCtrlPtr^.Output.monitor.FileUpdate.FileUpdate_Error   := 	enum_DriveUpdateError.FileClosedFailed;
			
			AxisCtrlPtr^.Output.monitor.FileUpdate.ErrorID:= FOE_Ctrl_UpdateFW.fbFileClose.nErrId;	
			UpdateFWState:=	12;	
		END_IF
		
	7:	
		// := 'Foe Read';
		
		FOE_Ctrl_UpdateFW.fbEcFoeLoad_0.bExecute:=TRUE;
		AxisCtrlPtr^.Output.Status.Drive.eUpdate_Staus:= enum_DriveUpdateStatus.UpDating;
		UpdateFWState:=UpdateFWState +1;
		
	8:		
	//	St_Elomo_Drive_List[Index].Progress:=FB_EcFoeLoad_0.nProgress;
		// := 'Load file';
		IF FOE_Ctrl_UpdateFW.fbEcFoeLoad_0.bBusy =FALSE THEN 		
			FOE_Ctrl_UpdateFW.fbEcFoeLoad_0.bExecute:=FALSE;		
			IF FOE_Ctrl_UpdateFW.fbEcFoeLoad_0.bError THEN 
				AxisCtrlPtr^.Output.Status.Drive.eUpdate_Staus :=	enum_DriveUpdateStatus.Error;				
				AxisCtrlPtr^.Output.monitor.FileUpdate.ErrorID:= FOE_Ctrl_UpdateFW.fbEcFoeLoad_0.nErrId;								
				AxisCtrlPtr^.Output.monitor.FileUpdate.FileUpdate_Error   := 	enum_DriveUpdateError.FileClosedFailed;
				UpdateFWState:=	130;
			ELSE
				UpdateFWState:=	100;
				AxisCtrlPtr^.Output.Status.Drive.eUpdate_Staus:= enum_DriveUpdateStatus.Updated;
			END_IF
						
		END_IF
		
	100:
		// := 'Load Done';

		

		Meth_DriveFWUpdate:=		TRUE;
	
END_CASE
//St_Elomo_Drive_List[Index].Status_String:=Local_Status_String[St_Elomo_Drive_List[Index].Update_Staus];
END_METHOD

METHOD Meth_FOE_fbCalls : BOOL
VAR_INPUT
END_VAR
FOE_Ctrl_Paramters.fbFileOpen(
	(*
	bExecute:= , 
	tTimeout:= , 
	bBusy=> , 
	bError=> , 
	nErrId=> , 
	hFile=> *)
); 



FOE_Ctrl_Paramters.fbFileClose(	
	hFile:= FOE_Ctrl_Paramters.hFile , 
	bExecute:= , 
	tTimeout:= , 
	bBusy=> , 
	bError=> , 
	nErrId=> );




FOE_Ctrl_Paramters.fbEcFoeLoad_0(	sNetId:=F_CreateAmsNetId(AxisCtrlPtr^.Input.Parameter.ecNetIdArr) , 
	nSlaveAddr:= AxisCtrlPtr^.Input.Parameter.Drive.EtherCatAddr, 
	sPathName:=FOE_Ctrl_Paramters.Foe_File_Path , 
	dwPass:= , 
	eMode:= eFoeMode_Write, 
	bExecute:= , 
	tTimeout:= , 
	bBusy=> , 
	bError=> , 
	nErrId=> , 
	cbLoad=> , 
	nProgress=> , 
	sInfo=> );
END_METHOD

METHOD PROTECTED Meth_Homing : BOOL
VAR_INPUT
	Execute   : BOOL;	
END_VAR
VAR_INST
	
	HomingState : INT;
END_VAR
IF HomeTrig.EDGEPOS(Execute) THEN

	Meth_Homing := FALSE;				

	HomingState := 1;
	HomingActive:= 		TRUE ;
	fbMC_Home.Execute:= FALSE;
END_IF


IF HomeTrig.EDGENEG(Execute) THEN
	
	HomingState := 0;
END_IF


CASE HomingState OF
	0:
		FB_EcCoeSdoWrite.bExecute := FALSE;
				
		Meth_CoEChangOperationMode(FALSE, eCaOpDriveModeOfOperation.CyclicSyncMode );
		Meth_ConfigHomeParamters(FALSE);
		HomeDirect(FALSE);
	1:	
		AxisCtrlPtr^.Input.Command.Power := FALSE;
		Meth_CoEChangOperationMode(FALSE,eCaOpDriveModeOfOperation.HomingMode);
		// Fix link problem
		IF strEcNetId= '' AND (AxisCtrlPtr^.Input.Parameter.ecNetIdArr[4]<>0 OR AxisCtrlPtr^.Input.Parameter.ecNetIdArr[5]<>0) THEN
			strEcNetId:= F_CreateAmsNetId(AxisCtrlPtr^.Input.Parameter.ecNetIdArr);
		END_IF	
		
		HomingState := 2;
	2:
		// changing mode to homing mode
		IF Meth_CoEChangOperationMode(TRUE,eCaOpDriveModeOfOperation.HomingMode) THEN			
			HomingState := 3;
		END_IF
	3://Config method and other params
	
		Homing_Ctrl_Params.HomingSWSpeed := LREAL_TO_UDINT( AxisCtrlPtr^.Input.Parameter.HomeOptions.stBasic.SwitchVelo);
		Homing_Ctrl_Params.HomingTrSpeed := LREAL_TO_UDINT( AxisCtrlPtr^.Input.Parameter.HomeOptions.stBasic.TriggerVelo);
		Homing_Ctrl_Params.HomingAcc     := LREAL_TO_UDINT( AxisCtrlPtr^.Input.Parameter.HomeOptions.stBasic.Acc);
		Homing_Ctrl_Params.HomingOffset  := LREAL_TO_DINT( AxisCtrlPtr^.Input.Parameter.HomeOptions.stBasic.HomeSetPos);
		IF Meth_ConfigHomeParamters(TRUE) THEN
			Meth_ConfigHomeParamters(FALSE);
			HomingState := 4;
		END_IF	
	4:
	
	//ETZ to Remove
		AxisCtrlPtr^.Input.Command.Power := TRUE;
		HomingState :=5;
		
	5: //Check homing attained				
		IF IsHomingAttained() THEN	
			AxisCtrlPtr^.Output.monitor.stAbsEncoder.BlockOffsetPosition := AxisCtrlPtr^.Output.monitor.ActPosition;
			fnLogMsg(ADR(LogMsg_0),LOG_INFO,'Block Pos %d ',LREAL_TO_DINT(AxisCtrlPtr^.Output.monitor.stAbsEncoder.BlockOffsetPosition),0,0);

			Meth_CoEChangOperationMode(FALSE,eCaOpDriveModeOfOperation.CyclicSyncMode);
			HomingState :=6;
		END_IF
	
	6: 
	
		fbMC_Home.HomingMode 					:= MC_Direct ;
		fbMC_Home.Options.ClearPositionLag 		:= TRUE ;
		IF MC_Block <> AxisCtrlPtr^.Input.Parameter.HomeOptions.stBasic.HomeMode THEN
			fbMC_Home.Position 						:= AxisCtrlPtr^.Input.Parameter.HomeOptions.stBasic.HomeSetPos;
			fnLogMsg(ADR(LogMsg_0),LOG_INFO,'Home Direct',0,0,0);
		ELSE
			fbMC_Home.Position 						:= AxisCtrlPtr^.Output.monitor.ActPosition;
			fnLogMsg(ADR(LogMsg_0),LOG_INFO,'Home Direct Set Act Pos For block',0,0,0);
		END_IF		
		fbMC_Home.Execute:= TRUE;
		HomingState := 7;

	
	7:
	
		IF fbMC_Home.Done THEN
			
			fbMC_Home.Execute := FALSE;
			Meth_CoEChangOperationMode(FALSE,eCaOpDriveModeOfOperation.CyclicSyncMode);
			HomingState := 8;
		END_IF

		
	

	8: 
	
		IF Meth_CoEChangOperationMode(TRUE,DINT_TO_SINT(eCaOpDriveModeOfOperation.CyclicSyncMode)) THEN
			Meth_CoEChangOperationMode(FALSE,eCaOpDriveModeOfOperation.CyclicSyncMode);
			Meth_Homing := TRUE;
		END_IF

		
END_CASE



{warning disable C0371}	

fbMC_Home(Axis:= AxisRef);

{warning restore C0371}
END_METHOD

METHOD Meth_InitVelKI : BOOL
VAR_INPUT
	Execute   : BOOL;
	Value	  : LREAL;
END_VAR

VAR_INST
	// Service Functions Variablea
	InitSctrlKITrigger : Trigger ;
	InitSctrlKIState   : SINT;
	
END_VAR
VAR
 
	
END_VAR
VAR_OUTPUT
	Error : BOOL;
END_VAR

IF InitSctrlKITrigger.EDGEPOS(Execute) THEN
	Meth_InitVelKI := FALSE;
	InitSctrlKIState := 1;
	EcCoeSdoWrite(FALSE);
END_IF


IF InitSctrlKITrigger.EDGENEG(Execute) THEN
	InitSctrlKIState := 0;
	Meth_InitVelKI := FALSE;
	EcCoeSdoWrite(FALSE);

END_IF

IF NOT AxisCtrlPtr^.Output.Status.Drive.ActiveHW THEN// SIM
	Meth_InitVelKI := TRUE;
ELSE

CASE InitSctrlKIState OF 
	0:
		Meth_InitVelKI := FALSE;
	1:
		
		CoeSdoRW.Input.Write.nIndex    := CoEDrive_Ctrl_Adr.KiSpeed.Index;	  
		CoeSdoRW.Input.Write.nSubIndex := CoEDrive_Ctrl_Adr.KiSpeed.SunIndex;
		RealValue := LREAL_TO_REAL(Value);
		CoeSdoRW.Input.Write.cbBufLen  := SIZEOF(RealValue);
	
		CoeSdoRW.Input.Write.pSrcBuf   :=   ADR(RealValue); 	 
	//	CoeSdoRW.Input.Write.cbBufLen  := SIZEOF(UdintValue)  ; 
		 
		IF EcCoeSdoWrite(TRUE , Error=> Error ) THEN
			EcCoeSdoWrite(FALSE , Error=> Error );
			InitSctrlKIState := InitSctrlKIState +1;
		END_IF
	
	2:
		Meth_InitVelKI := TRUE;

END_CASE
END_IF
END_METHOD

METHOD Meth_InitVelKP : BOOL
VAR_INPUT
	Execute   : BOOL;
	Value	  : LREAL;
END_VAR

VAR_INST
	//
	InitSctrlKPTrigger : Trigger ;
	InitSctrlKPState 	 : SINT;		
	
END_VAR

VAR


END_VAR

VAR_OUTPUT
	Error : BOOL;
END_VAR

IF InitSctrlKPTrigger.EDGEPOS(Execute) THEN
	Meth_InitVelKP := FALSE;
	InitSctrlKPState := 1;
	Error := FALSE;
	EcCoeSdoWrite(FALSE);
END_IF


IF InitSctrlKPTrigger.EDGENEG(Execute) THEN
	InitSctrlKPState := 0;
	Meth_InitVelKP := FALSE;
	EcCoeSdoWrite(FALSE);

END_IF
IF NOT AxisCtrlPtr^.Output.Status.Drive.ActiveHW THEN// SIM
	Meth_InitVelKP := TRUE;
ELSE


CASE InitSctrlKPState OF 
 
	1:
		
		CoeSdoRW.Input.Write.nIndex    := CoEDrive_Ctrl_Adr.KpSpeed.Index;	  
		CoeSdoRW.Input.Write.nSubIndex := CoEDrive_Ctrl_Adr.KpSpeed.SunIndex;
		RealValue := LREAL_TO_REAL(Value);
		CoeSdoRW.Input.Write.cbBufLen  := SIZEOF(RealValue);
	
		CoeSdoRW.Input.Write.pSrcBuf   :=   ADR(RealValue); 	 
	//	CoeSdoRW.Input.Write.cbBufLen  := SIZEOF(UdintValue)  ; 
		 
		IF EcCoeSdoWrite(TRUE , Error=> Error ) THEN
			EcCoeSdoWrite(FALSE , Error=> Error );
			InitSctrlKPState := InitSctrlKPState +1;
		END_IF
	
	2:
		Meth_InitVelKP := TRUE;

END_CASE
END_IF
END_METHOD

METHOD Meth_ReadObj : BOOL
VAR_INPUT
	Execute   : BOOL;
	Object	  : enumMotionObject;
	
END_VAR

VAR_INST
	ReadObjState  : USINT;
	ReadObjTrig: Trigger;
	IsRealValue:  BOOL;
	 
END_VAR
VAR
 TempValue : DINT;
	
END_VAR
VAR_OUTPUT
	Error : BOOL;
	Value : LREAL;
END_VAR

IF ReadObjTrig.EDGEPOS(Execute) THEN
	Meth_ReadObj := FALSE;
	ReadObjState := 1;
END_IF


IF ReadObjTrig.EDGENEG(Execute) THEN
	ReadObjState := 0;
	Meth_ReadObj := FALSE;
	EcCoeSdoRead(FALSE);

END_IF

IF NOT AxisCtrlPtr^.Output.Status.Drive.ActiveHW THEN// SIM
	Meth_ReadObj := TRUE;
ELSE

CASE ReadObjState OF 
	 
	1:
		CASE Object OF
			enumMotionObject.OPERATION_MODE :
			
				CoeSdoRW.Input.Read.nIndex		 := CoEDrive_Ctrl_Adr.OperationMode.Index;
				CoeSdoRW.Input.Read.nSubIndex	 := CoEDrive_Ctrl_Adr.OperationMode.SunIndex ;
				CoeSdoRW.Input.Read.cbBufLen	 := CoEDrive_Ctrl_Adr.OperationMode.Size ;
				
				IsRealValue 					 := CoEDrive_Ctrl_Adr.OperationMode.IsReal;
				
			enumMotionObject.VEL_KI:

				CoeSdoRW.Input.Read.nIndex		 := CoEDrive_Ctrl_Adr.KISpeed.Index;
				CoeSdoRW.Input.Read.nSubIndex	 := CoEDrive_Ctrl_Adr.KISpeed.SunIndex ;
				CoeSdoRW.Input.Read.cbBufLen	 := CoEDrive_Ctrl_Adr.KISpeed.Size ;		

				IsRealValue 					 := CoEDrive_Ctrl_Adr.KISpeed.IsReal;
		
			enumMotionObject.VEL_KP:
			
				CoeSdoRW.Input.Read.nIndex		 := CoEDrive_Ctrl_Adr.KpSpeed.Index;
				CoeSdoRW.Input.Read.nSubIndex	 := CoEDrive_Ctrl_Adr.KpSpeed.SunIndex ;
				CoeSdoRW.Input.Read.cbBufLen	 := CoEDrive_Ctrl_Adr.KpSpeed.Size ;
				
				IsRealValue 					 := CoEDrive_Ctrl_Adr.KpSpeed.IsReal;
				
			enumMotionObject.TORQUE_OFFSET:
			
				CoeSdoRW.Input.Read.nIndex		 := CoEDrive_Ctrl_Adr.TorqueOffset.Index;
				CoeSdoRW.Input.Read.nSubIndex	 := CoEDrive_Ctrl_Adr.TorqueOffset.SunIndex ;
				CoeSdoRW.Input.Read.cbBufLen	 := CoEDrive_Ctrl_Adr.TorqueOffset.Size ;
				
				IsRealValue 					 := CoEDrive_Ctrl_Adr.TorqueOffset.IsReal;
				
			enumMotionObject.MAX_TORQUE:	
				CoeSdoRW.Input.Read.nIndex		 := CoEDrive_Ctrl_Adr.MaxTorque.Index;
				CoeSdoRW.Input.Read.nSubIndex	 := CoEDrive_Ctrl_Adr.MaxTorque.SunIndex;
				CoeSdoRW.Input.Read.cbBufLen	 := CoEDrive_Ctrl_Adr.MaxTorque.Size ;
				
				IsRealValue 					 := CoEDrive_Ctrl_Adr.MaxTorque.IsReal;
				
			enumMotionobject.GAIN_SCHEDULE:		
				CoeSdoRW.Input.Read.nIndex		 := CoEDrive_Ctrl_Adr.GainScheduler.Index;
				CoeSdoRW.Input.Read.nSubIndex	 := CoEDrive_Ctrl_Adr.GainScheduler.SunIndex;
				CoeSdoRW.Input.Read.cbBufLen	 := CoEDrive_Ctrl_Adr.GainScheduler.Size ;				
				IsRealValue 					 := CoEDrive_Ctrl_Adr.GainScheduler.IsReal;
			
			enumMotionobject.ACC_CLOSE_POS_ERR:
				CoeSdoRW.Input.Read.nIndex		 := CoEDrive_Ctrl_Adr.AccClosePosErr.Index;
				CoeSdoRW.Input.Read.nSubIndex	 := CoEDrive_Ctrl_Adr.AccClosePosErr.SunIndex;
				CoeSdoRW.Input.Read.cbBufLen	 := CoEDrive_Ctrl_Adr.AccClosePosErr.Size ;				
				IsRealValue 					 := CoEDrive_Ctrl_Adr.AccClosePosErr.IsReal;
			enumMotionobject.DC_VOLATAGE:
				CoeSdoRW.Input.Read.nIndex		 := CoEDrive_Ctrl_Adr.DCVoltage.Index;
				CoeSdoRW.Input.Read.nSubIndex	 := CoEDrive_Ctrl_Adr.DCVoltage.SunIndex;
				CoeSdoRW.Input.Read.cbBufLen	 := CoEDrive_Ctrl_Adr.DCVoltage.Size ;				
				IsRealValue 					 := CoEDrive_Ctrl_Adr.DCVoltage.IsReal;
			
				
				
		END_CASE
		
		IF IsRealValue THEN
			CoeSdoRW.Input.Read.pDstBuf   :=   ADR(RealValue);
		ELSE
			
			CASE CoeSdoRW.Input.Read.cbBufLen OF 
				1:
					CoeSdoRW.Input.Read.pDstBuf   :=   ADR(UsintValue);
				2:
					CoeSdoRW.Input.Read.pDstBuf   :=   ADR(UintValue );
				4:
				
					CoeSdoRW.Input.Read.pDstBuf   :=   ADR(UdintValue);
				8:
					CoeSdoRW.Input.Read.pDstBuf   :=   ADR(Ulong);
				
	
			END_CASE		
 		END_IF 
		  
		IF NOT  CoeSdoRW.Output.Read.Busy THEN
			EcCoeSdoRead (FALSE  ); 			
			ReadObjState := ReadObjState +1;
		END_IF	

	
	2:
			IF EcCoeSdoRead (TRUE  ) THEN
				
				 
				IF IsRealValue THEN
					Value := RealValue;
				ELSE
					CASE CoeSdoRW.Input.Read.cbBufLen OF 
						1:
							Value   :=   USINT_TO_LREAL(UsintValue);
						2:
							Value   :=   UINT_TO_LREAL(UintValue) ;
						4:				
							Value   :=   UDINT_TO_REAL(UdintValue);
						8:
							Value  :=   ULINT_TO_LREAL(Ulong);	
					END_CASE
				END_IF
			

				
			
			
			
			IF  Object = enumMotionObject.TORQUE_OFFSET OR
				Object = enumMotionObject.MAX_TORQUE THEN
				Value := DriveUnitsTorqueToRealValue(Value);
	
			END_IF	
			LogText := 'Meth_ReadObj Value';
			LogText	:= CONCAT(LogText, 'Index 0x');
			LogText	:= CONCAT(LogText, UDINT_TO_HEX_STRING(CoeSdoRW.Input.Read.nIndex));
			LogText	:= CONCAT(LogText, ', SubIndex=');
			LogText	:= CONCAT(LogText, UDINT_TO_STRING(CoeSdoRW.Input.Read.nSubIndex));
			LogText	:= CONCAT(LogText, ', Value =');
			
			IF IsRealValue THEN
				TempValue := TO_DINT(Value* 1000);	
				LogText	:= CONCAT(LogText, ',(Real*1000) ');			
			ELSE	
 				TempValue := TO_DINT(Value);	
			END_IF
			LogText	:= CONCAT(LogText, DINT_TO_STRING(TempValue));
			fnLogMsg(ADR(LogMsg_0),LOG_INFO,LogText, 0,0,0);
		
			ReadObjState := ReadObjState +1;
			
			Meth_ReadObj := TRUE;
			
		END_IF
	
	
	3:
		Meth_ReadObj := TRUE;
		

END_CASE
END_IF
END_METHOD

METHOD Meth_TorqueInDriveUnits : LREAL
VAR_INPUT
	
	Torque: LREAL;	

END_VAR
Meth_TorqueInDriveUnits := Torque;
END_METHOD

METHOD Meth_UpdateDriveParams : BOOL
VAR_INPUT
	Execute:		BOOL;
END_VAR
VAR_INST
	UpdateDriveParamsTrig  : 	Trigger;
	UpdateDriveParamsState : INT;
	
	 
END_VAR
IF UpdateDriveParamsTrig.EDGEPOS(Execute) THEN
	
	UpdateDriveParamsState := 0;
	AxisCtrlPtr^.Output.Status.Drive.eUpdate_Staus := enum_DriveUpdateStatus.NoAction;
	AxisCtrlPtr^.Output.monitor.FileUpdate.FileUpdate_Error   := 	enum_DriveUpdateError.NoError;
	AxisCtrlPtr^.Output.monitor.FileUpdate.ErrorID := 0;
END_IF



CASE UpdateDriveParamsState OF 
	0://init -wait	

		
		UpdateDriveParamsState:=UpdateDriveParamsState +1;
	
	1://read Version Drive Param Version	
		// := 'Read Version';			
							
		CoeSdoRW.Input.Read.nIndex 	  := CoEDrive_Ctrl_Adr.ParamsVersionObj.Index; 
		CoeSdoRW.Input.Read.nSubIndex := CoEDrive_Ctrl_Adr.ParamsVersionObj.SunIndex;
		CoeSdoRW.Input.Read.pDstBuf	  := ADR(FOE_Ctrl_Paramters.Version_From_Drive);
 		CoeSdoRW.Input.Read.cbBufLen  := SIZEOF(FOE_Ctrl_Paramters.Version_From_Drive);  

		FOE_Ctrl_Paramters.fbFileOpen.bExecute    := FALSE;
		FOE_Ctrl_Paramters.fbFileClose.bExecute   := FALSE;
		FOE_Ctrl_Paramters.fbEcFoeLoad_0.bExecute := FALSE;
		EcCoeSdoRead(FALSE);
		FOE_Ctrl_Paramters.Foe_File_Path:=AxisCtrlPtr^.Input.Parameter.Drive.sFoeParams_Path;
		UpdateDriveParamsState:= UpdateDriveParamsState +1;

		
	2://Download to Drive 
		// := 'Download to Drive';
		IF EcCoeSdoRead(TRUE) THEN		
  				
			AxisCtrlPtr^.Output.Status.Drive.ParamVer:=	FOE_Ctrl_Paramters.Version_From_Drive;	
			IF AxisCtrlPtr^.Output.Status.Drive.ParamVer <> AxisCtrlPtr^.Input.Parameter.Drive.LatestParamVer THEN				
				AxisCtrlPtr^.Output.Status.Drive.eUpdate_Staus:= enum_DriveUpdateStatus.Checking;
				UpdateDriveParamsState:=UpdateDriveParamsState +1;
			ELSE
				AxisCtrlPtr^.Output.Status.Drive.eUpdate_Staus:= enum_DriveUpdateStatus.Updated;
				UpdateDriveParamsState:=	100;										
			END_IF
						
		END_IF
		
	3: 
		
						
		FOE_Ctrl_Paramters.fbFileOpen.sNetId		:= ''; 
		FOE_Ctrl_Paramters.fbFileOpen.sPathName		:=FOE_Ctrl_Paramters.Foe_File_Path; 
		FOE_Ctrl_Paramters.fbFileOpen.nMode			:=FOPEN_MODEREAD; 
		FOE_Ctrl_Paramters.fbFileOpen.ePath			:=PATH_GENERIC ;
		
		FOE_Ctrl_Paramters.fbFileOpen.bExecute:=	TRUE; 

		UpdateDriveParamsState:=UpdateDriveParamsState +1;
	4:
		//Check Valid file Path
		// := 'Cheack Valid Path';
		
		IF FOE_Ctrl_Paramters.fbFileOpen.bBusy =FALSE AND FOE_Ctrl_Paramters.fbFileOpen.bError =FALSE THEN 
			FOE_Ctrl_Paramters.hFile := FOE_Ctrl_Paramters.fbFileOpen.hFile;
			FOE_Ctrl_Paramters.fbFileOpen.bExecute:=	FALSE;
			UpdateDriveParamsState:=UpdateDriveParamsState +1;
			
			
			
			
		ELSIF FOE_Ctrl_Paramters.fbFileOpen.bError =TRUE THEN 
			AxisCtrlPtr^.Output.Status.Drive.eUpdate_Staus 			  :=	enum_DriveUpdateStatus.Error;
			AxisCtrlPtr^.Output.monitor.FileUpdate.FileUpdate_Error   := 	enum_DriveUpdateError.FileNotFound;
			AxisCtrlPtr^.Output.monitor.FileUpdate.ErrorID 			  :=    FOE_Ctrl_Paramters.fbFileOpen.nErrId;
			UpdateDriveParamsState:=	11;				
		END_IF	
	5:
			FOE_Ctrl_Paramters.fbFileClose.bExecute:=	TRUE;	
			UpdateDriveParamsState:=UpdateDriveParamsState +1;
	6:	
		// := 'Close path';
		
		IF FOE_Ctrl_Paramters.fbFileClose.bBusy =FALSE AND FOE_Ctrl_Paramters.fbFileClose.bError =FALSE THEN 
			FOE_Ctrl_Paramters.fbFileClose.bExecute:=FALSE;	
			UpdateDriveParamsState:=UpdateDriveParamsState +1;

			
	
		ELSIF FOE_Ctrl_Paramters.fbFileClose.bError =TRUE THEN 
			AxisCtrlPtr^.Output.Status.Drive.eUpdate_Staus :=	enum_DriveUpdateStatus.Error;
			AxisCtrlPtr^.Output.monitor.FileUpdate.FileUpdate_Error   := 	enum_DriveUpdateError.FileClosedFailed;
			
			AxisCtrlPtr^.Output.monitor.FileUpdate.ErrorID:= FOE_Ctrl_Paramters.fbFileClose.nErrId;	
			UpdateDriveParamsState:=	12;	
		END_IF
		
	7:	
		// := 'Foe Read';
		
		FOE_Ctrl_Paramters.fbEcFoeLoad_0.bExecute:=TRUE;
		AxisCtrlPtr^.Output.Status.Drive.eUpdate_Staus:= enum_DriveUpdateStatus.UpDating;
		UpdateDriveParamsState:=UpdateDriveParamsState +1;
		
	8:		
	//	St_Elomo_Drive_List[Index].Progress:=FB_EcFoeLoad_0.nProgress;
		// := 'Load file';
		IF FOE_Ctrl_Paramters.fbEcFoeLoad_0.bBusy =FALSE THEN 		
			FOE_Ctrl_Paramters.fbEcFoeLoad_0.bExecute:=FALSE;		
			IF FOE_Ctrl_Paramters.fbEcFoeLoad_0.bError THEN 
				AxisCtrlPtr^.Output.Status.Drive.eUpdate_Staus :=	enum_DriveUpdateStatus.Error;				
				AxisCtrlPtr^.Output.monitor.FileUpdate.ErrorID:= FOE_Ctrl_Paramters.fbEcFoeLoad_0.nErrId;								
				AxisCtrlPtr^.Output.monitor.FileUpdate.FileUpdate_Error   := 	enum_DriveUpdateError.FileClosedFailed;
				UpdateDriveParamsState:=	130;
			ELSE
				UpdateDriveParamsState:=	100;
				AxisCtrlPtr^.Output.Status.Drive.eUpdate_Staus:= enum_DriveUpdateStatus.Updated;
			END_IF
						
		END_IF
		
	100:
		// := 'Load Done';

		

		Meth_UpdateDriveParams:=		TRUE;
	
END_CASE
//St_Elomo_Drive_List[Index].Status_String:=Local_Status_String[St_Elomo_Drive_List[Index].Update_Staus];
END_METHOD

METHOD Meth_WriteObj : BOOL
VAR_INPUT
	Execute   : BOOL;
	Object	  : enumMotionObject;
	Value	  : LREAL;
	
END_VAR


VAR


	
	TempValue: DINT;
END_VAR
VAR_INST
	WriteObjState  : USINT;
	WriteObjTrig: Trigger;
	IsRealValue:  BOOL;
END_VAR


VAR_OUTPUT
	Error : BOOL;
END_VAR

IF WriteObjTrig.EDGEPOS(Execute) THEN
	Meth_WriteObj := FALSE;
	WriteObjState := 1;
END_IF


IF WriteObjTrig.EDGENEG(Execute) THEN
	WriteObjState := 0;
	Meth_WriteObj := FALSE;
	EcCoeSdoWrite(FALSE);

END_IF

IF NOT AxisCtrlPtr^.Output.Status.Drive.ActiveHW THEN// SIM
	Meth_WriteObj := TRUE;	
ELSE

CASE WriteObjState OF 
	 
	1:
		
		CASE Object OF
			enumMotionObject.OPERATION_MODE :
			
				CoeSdoRW.Input.Write.nIndex		 := CoEDrive_Ctrl_Adr.OperationMode.Index;
				CoeSdoRW.Input.Write.nSubIndex	 := CoEDrive_Ctrl_Adr.OperationMode.SunIndex ;
				CoeSdoRW.Input.Write.cbBufLen	 := CoEDrive_Ctrl_Adr.OperationMode.Size ;
				IsRealValue 					 := CoEDrive_Ctrl_Adr.OperationMode.IsReal;
			enumMotionObject.VEL_KI:

				CoeSdoRW.Input.Write.nIndex		 := CoEDrive_Ctrl_Adr.KISpeed.Index;
				CoeSdoRW.Input.Write.nSubIndex	 := CoEDrive_Ctrl_Adr.KISpeed.SunIndex ;
				CoeSdoRW.Input.Write.cbBufLen	 := CoEDrive_Ctrl_Adr.KISpeed.Size ;	
				IsRealValue 					 := CoEDrive_Ctrl_Adr.KISpeed.IsReal;			
			enumMotionObject.VEL_KP:
			
				CoeSdoRW.Input.Write.nIndex		 := CoEDrive_Ctrl_Adr.KpSpeed.Index;
				CoeSdoRW.Input.Write.nSubIndex	 := CoEDrive_Ctrl_Adr.KpSpeed.SunIndex ;
				CoeSdoRW.Input.Write.cbBufLen	 := CoEDrive_Ctrl_Adr.KpSpeed.Size ;
				IsRealValue 					 := CoEDrive_Ctrl_Adr.KpSpeed.IsReal;
			enumMotionObject.TORQUE_OFFSET:
			
				CoeSdoRW.Input.Write.nIndex		 := CoEDrive_Ctrl_Adr.TorqueOffset.Index;
				CoeSdoRW.Input.Write.nSubIndex	 := CoEDrive_Ctrl_Adr.TorqueOffset.SunIndex ;
				CoeSdoRW.Input.Write.cbBufLen	 := CoEDrive_Ctrl_Adr.TorqueOffset.Size ;
				IsRealValue 					 := CoEDrive_Ctrl_Adr.TorqueOffset.IsReal;
				Value := Meth_TorqueInDriveUnits( Value);
				
			enumMotionObject.MAX_TORQUE:	
				CoeSdoRW.Input.Write.nIndex		 := CoEDrive_Ctrl_Adr.MaxTorque.Index;
				CoeSdoRW.Input.Write.nSubIndex	 := CoEDrive_Ctrl_Adr.MaxTorque.SunIndex;
				CoeSdoRW.Input.Write.cbBufLen	 := CoEDrive_Ctrl_Adr.MaxTorque.Size ;
				IsRealValue 					 := CoEDrive_Ctrl_Adr.MaxTorque.IsReal;
				Value := Meth_TorqueInDriveUnits( Value);
				
			enumMotionObject.GAIN_SCHEDULE:
				CoeSdoRW.Input.Write.nIndex		 := CoEDrive_Ctrl_Adr.GainScheduler.Index;
				CoeSdoRW.Input.Write.nSubIndex	 := CoEDrive_Ctrl_Adr.GainScheduler.SunIndex;
				CoeSdoRW.Input.Write.cbBufLen	 := CoEDrive_Ctrl_Adr.GainScheduler.Size ;
				IsRealValue 					 := CoEDrive_Ctrl_Adr.GainScheduler.IsReal;
				
			enumMotionObject.ACC_CLOSE_POS_ERR:
				CoeSdoRW.Input.Write.nIndex		 := CoEDrive_Ctrl_Adr.AccClosePosErr.Index;
				CoeSdoRW.Input.Write.nSubIndex	 := CoEDrive_Ctrl_Adr.AccClosePosErr.SunIndex;
				CoeSdoRW.Input.Write.cbBufLen	 := CoEDrive_Ctrl_Adr.AccClosePosErr.Size ;
				IsRealValue 					 := CoEDrive_Ctrl_Adr.AccClosePosErr.IsReal;		
				
		END_CASE
		
		IF IsRealValue THEN
				RealValue := LREAL_TO_REAL(Value);
				CoeSdoRW.Input.Write.pSrcBuf   :=   ADR(RealValue);			
		ELSE
			CASE CoeSdoRW.Input.Write.cbBufLen OF 
				1:
					UsintValue := LREAL_TO_USINT(Value);
					CoeSdoRW.Input.Write.pSrcBuf   :=   ADR(UsintValue);
				2:
					UintValue := LREAL_TO_UINT(Value);
					CoeSdoRW.Input.Write.pSrcBuf   :=   ADR(UintValue );
				4:
					UdintValue := LREAL_TO_UDINT(Value);
					CoeSdoRW.Input.Write.pSrcBuf   :=   ADR(UdintValue);
				8:
					Ulong := LREAL_TO_ULINT(Value);
					CoeSdoRW.Input.Write.pSrcBuf   :=   ADR(Ulong);
				
			END_CASE		
		END_IF
		IF NOT CoeSdoRW.Output.Write.Busy THEN			 
			EcCoeSdoWrite(FALSE , Error=> Error );
	
			
			LogText := 'Meth_WriteObj Value';
			LogText	:= CONCAT(LogText, 'Index 0x');
			LogText	:= CONCAT(LogText, UDINT_TO_HEX_STRING(CoeSdoRW.Input.Write.nIndex));
			LogText	:= CONCAT(LogText, ', SubIndex=');
			LogText	:= CONCAT(LogText, UDINT_TO_STRING(CoeSdoRW.Input.Write.nSubIndex));
			LogText	:= CONCAT(LogText, ', Value =');
			
			IF IsRealValue THEN
				LogText	:= CONCAT(LogText, ',(Real*1000) ');
				TempValue := TO_DINT(Value* 1000);				
			ELSE	
 				TempValue := TO_DINT(Value);	
			END_IF
			LogText	:= CONCAT(LogText, DINT_TO_STRING(TempValue));
			fnLogMsg(ADR(LogMsg_0),LOG_INFO,LogText, 0,0,0);

			



			
			WriteObjState := WriteObjState +1;
		END_IF	
		
	2:
		IF EcCoeSdoWrite(TRUE , Error=> Error ) THEN
			EcCoeSdoWrite(FALSE , Error=> Error );
			WriteObjState := WriteObjState +1;
		END_IF
	
	3:
		
		Meth_WriteObj := TRUE;

END_CASE
END_IF
END_METHOD

METHOD ReadActualCurrent : LREAL
VAR_INPUT
END_VAR
VAR_INST
		
END_VAR

AxisCtrlPtr^.Output.monitor.ActualCurrent	:=  ( (THIS^.io_ActualCurrent) / 1000.0)/SQRT(2.0) * (UDINT_TO_LREAL(CoeRead_RatedCurrent) / 1000.0);

//AxisCtrlPtr^.Output.monitor.ActualCurrent	:=  ( (THIS^.io_ActualCurrent) / 1000.0) * AxisCtrlPtr^.Input.Parameter.RatedCurrent;
END_METHOD

METHOD ReadActualTorque : LREAL
VAR_INPUT
END_VAR

//AxisCtrlPtr^.Output.monitor.ActualTorque	:=  (INT_TO_LREAL(THIS^.io_ActualTorque) / 1000.0)/SQRT(2.0) * (UDINT_TO_LREAL(CoeRead_RatedTorque) / 1000.0);

AxisCtrlPtr^.Output.monitor.ActualTorque	:=  ((THIS^.io_ActualTorque) / 1000.0) * AxisCtrlPtr^.Input.Parameter.Ratedtorque;
END_METHOD

METHOD ReadDcVoltage : BOOL
VAR_INPUT
END_VAR
VAR_INST
	ReadDcTimer : TON;
END_VAR
	ReadDcTimer.IN := TRUE;
	ReadDcTimer.PT := T#20S;
		
	IF ReadDcTimer.Q THEN			 
			ReadDcTimer.IN := FALSE;

 		IF  Meth_ReadObj(TRUE, enumMotionObject.DC_VOLATAGE, Value =>LRealValue, Error =>ReadObjError ) THEN
					AxisCtrlPtr^.Output.monitor.ActualDC :=    RealValue;
					Meth_ReadObj(FALSE, enumMotionObject.DC_VOLATAGE  );											
		END_IF
	END_IF
	
	ReadDcTimer();
END_METHOD

METHOD ReadInitDriveParID : BOOL
VAR_INPUT
	bStart : BOOL;
END_VAR

VAR_INST
	ExecuteTrig: 		Trigger;
	State_InitSpecific: INT;
END_VAR

IF ExecuteTrig.EDGEPOS(bStart) THEN
	ReadInitDriveParID		:= FALSE;
	State_InitSpecific	:= 1;		
END_IF

IF ExecuteTrig.EDGENEG(bStart) THEN
	State_InitSpecific	:= 0;	
	ReadInitDriveParID		:= FALSE;
END_IF

CASE State_InitSpecific OF

	 
	1:
		EcCoeSdoRead(FALSE);
		CoeSdoRW.Input.Read.nIndex		:= DINT_TO_WORD(eDS402DriveParID.MotorRatedCurrent);
		CoeSdoRW.Input.Read.nSubIndex	:= 0;
		CoeSdoRW.Input.Read.pDstBuf		:= ADR(CoeRead_RatedCurrent);
		CoeSdoRW.Input.Read.cbBufLen	:= SIZEOF(CoeRead_RatedCurrent);
		State_InitSpecific	:= 2;
		
	2:
		IF EcCoeSdoRead(TRUE) THEN	
			State_InitSpecific	:= 3;
		END_IF
		
	3:
		EcCoeSdoRead(FALSE);
		CoeSdoRW.Input.Read.nIndex		:= DINT_TO_WORD(eDS402DriveParID.MotorRatedTorque);
		CoeSdoRW.Input.Read.nSubIndex	:= 0;
		CoeSdoRW.Input.Read.pDstBuf		:= ADR(CoeRead_RatedTorque);
		CoeSdoRW.Input.Read.cbBufLen	:= SIZEOF(CoeRead_RatedTorque);
		State_InitSpecific	:= 4;
		
	4:
		IF EcCoeSdoRead(TRUE) THEN
			AxisCtrlPtr^.Input.Parameter.RatedCurrent	:= UDINT_TO_LREAL(CoeRead_RatedCurrent) / 1000.0;
			AxisCtrlPtr^.Input.Parameter.Ratedtorque	:= UDINT_TO_LREAL(CoeRead_RatedTorque) / 100.0;
			ReadInitDriveParID		:= TRUE;	
			State_InitSpecific	:= 0;
		END_IF
		
		
 
		
END_CASE
END_METHOD

END_FUNCTION_BLOCK

// ---- POUs/Lib/Motion/CanOpenAxis/Elmo/FB_ElmoIOsHandle.TcPOU
FUNCTION_BLOCK FB_ElmoIOsHandle
VAR_INPUT
	DigIn:		DINT;		
END_VAR
VAR_OUTPUT
	bEnable:			BOOL;
	bDriveHomeSignal:	BOOL;
	arrDigIn:			ARRAY[1..10] OF BOOL;		
END_VAR
VAR
END_VAR

bEnable:=			DigIn.3;
bDriveHomeSignal:= 	DigIn.2;
arrDigIn[1]:=		DigIn.16;		
arrDigIn[2]:=		DigIn.17;		
arrDigIn[3]:=		DigIn.18;		
arrDigIn[4]:=		DigIn.19;			
arrDigIn[5]:=		DigIn.20;			
arrDigIn[6]:=		DigIn.21;			
arrDigIn[7]:=		DigIn.22;	
arrDigIn[8]:=		DigIn.23;
arrDigIn[9]:=		DigIn.24;
arrDigIn[10]:=		DigIn.25;

END_FUNCTION_BLOCK

// ---- POUs/Lib/Motion/FailureRport/Motor/MotorFailureReport_FB.TcPOU
FUNCTION_BLOCK MotorFailureReport_FB
VAR_INPUT
	AxisCtrlPtr			: POINTER TO Basic_axis_typ ;
	StationID 			: eStationNo;
	
	(*Ref_ev_MOTOR_POSITION   : REFERENCE TO ev_MOTOR_POSITION_ERROR REF= ev_MOTOR_POSITION_ERROR;
	Ref_ev_MOTOR_Speed      : REFERENCE TO ev_MOTOR_SPEED_ERROR    REF= ev_MOTOR_SPEED_ERROR;	
	Ref_ev_HOME_NOT_FOUND   : REFERENCE TO ev_MOTOR_HOME_NOT_FOUND REF= ev_MOTOR_HOME_NOT_FOUND;
	Ref_ev_OVER_CURRENT     : REFERENCE TO ev_MOTOR_OVER_CURRENT   REF= ev_MOTOR_OVER_CURRENT;

	Ref_ev_MOTOR_OVER_TEMP      : REFERENCE TO  ev_MOTOR_OVER_TEMP        REF= ev_MOTOR_OVER_TEMP;
	Ref_ev_MOTOR_FEEDBACK_ERROR : REFERENCE TO	ev_MOTOR_FEEDBACK_ERROR   REF=  ev_MOTOR_FEEDBACK_ERROR ;
	Ref_ev_MOTOR_GENERAL_ERROR 	: REFERENCE TO	ev_MOTOR_GENERAL_ERROR    REF=  ev_MOTOR_GENERAL_ERROR ;
	Ref_ev_MOTOR_STALLED		: REFERENCE TO  ev_MOTOR_STALLED          REF=  ev_MOTOR_STALLED;
	Ref_ev_MOTOR_SUPPLY_ERROR 	: REFERENCE TO	ev_MOTOR_SUPPLY_ERROR     REF=  ev_MOTOR_SUPPLY_ERROR ;
 	Ref_ev_PLC_ILLEGAL_MSG  	: REFERENCE TO	ev_PLC_ILLEGAL_MSG        REF= 	ev_PLC_ILLEGAL_MSG  ;
	Ref_ev_PLC_ILLEGAL_PARAM 	: REFERENCE TO	ev_PLC_ILLEGAL_PARAM      REF= 	ev_PLC_ILLEGAL_PARAM ;
	Ref_ev_Drive_Not_Enabled 	: REFERENCE TO  ev_MOTOR_DRIVE_NOT_ENABLED REF= 	ev_MOTOR_DRIVE_NOT_ENABLED ;
	
	Ref_ev_DRIVE_NOT_READY    	: REFERENCE TO	ev_MOTOR_DRIVE_NOT_READY  REF= 	ev_MOTOR_DRIVE_NOT_READY ;
	Ref_ev_Drive_ComError		: REFERENCE TO  ev_MOTOR_DRIVE_COM_ERROR  REF= 	ev_MOTOR_DRIVE_COM_ERROR ;
	Ref_ev_BRAKE_RESISTOR_ERROR : REFERENCE TO  ev_BRAKE_RESISTOR_ERROR   REF= 	ev_BRAKE_RESISTOR_ERROR ;
	*)
	

                                                                            
	                                                                        


	
	
END_VAR
VAR
	LastErrorId			: UDINT;
	PrevErrorId			: UDINT;
	AxisLastErrorCount  : UDINT := 0;
	Pop_Delay	 		: TON;
	ErrorID_Delay 		: TON;
	lastEventID: enumMotorEvents;
	MotorErrorQ			: Queue;
	QErrorCounter       : UDINT;
	//
	LogMsgInit          : BOOL := TRUE;
	LogMsg_0 			: LogMsg ;
	//Get old events from Q
	PrevMotorEvents		: Eh_ErrorEntry_typ;
	ThreadName		    : STRING[20];	
	fbPrgmBasic			:FB_PrgmBasic;
	
	//EventParameters:EventParam_Typ;	
	//EventHeader:EventHeader_Typ;	
	
END_VAR

//Classifier
//Method






IF AxisCtrlPtr <> 0 THEN
		
	IF LogMsgInit THEN      
		LogMsgInit := FALSE ;
		ThreadName := AxisCtrlPtr^.Input.Parameter.ThreadName;
		CONCAT(  ThreadName,'Re');
		fnLogMsgInit(ADR(LogMsg_0), ThreadName, ADR(LogGlobalArray), ADR(CONST_ZERO));
		LogMsg_0.Enable:= 		TRUE;
	END_IF

	IF AxisCtrlPtr^.Output.Error.ErrorCount > 0 AND AxisCtrlPtr^.Input.Command.ErrorAcknowledge = FALSE THEN
		ErrorID_Delay.PT := T#25MS ;	
		Pop_Delay.IN := TRUE;	
			
			
	END_IF
	
	
	IF Pop_Delay.Q THEN
		Pop_Delay.IN := FALSE;
		AxisCtrlPtr^.Input.Command.ErrorAcknowledge := TRUE;
	END_IF	
	Pop_Delay();
	
	//Add code for clear error	
	ErrorID_Delay.IN := AxisCtrlPtr^.Output.Error.ErrorCount  = 0 AND AxisCtrlPtr^.Output.Status.FAULT ;
	ErrorID_Delay.PT := T#100MS ;
	ErrorID_Delay();
						
	IF ErrorID_Delay.Q THEN
		
		AxisCtrlPtr^.Input.Command.ClearFault := TRUE;
		
	END_IF
	

	//Check if there is new error
	IF AxisCtrlPtr^.Output.Error.fbErrorHandler.EntriesCount <> 0 AND
	  lastEventID<> AxisCtrlPtr^.Output.Error.ErrorEntry.MotorEvents AND 
	  AxisCtrlPtr^.Output.Error.ErrorEntry.MotorEvents <> enumMotorEvents.NoEvents THEN		
		
		AxisLastErrorCount := AxisCtrlPtr^.Output.Error.fbErrorHandler.EntriesCount;
	 	
		IF Meth_GetEvent( AxisCtrlPtr^.Output.Error.ErrorEntry ) = FALSE THEN
			
			MotorErrorQ.Enqueue(ADR(AxisCtrlPtr^.Output.Error.ErrorEntry),SIZEOF(Eh_ErrorEntry_typ));	
			IF AxisCtrlPtr^.Input.Parameter.pFlowID <> 0 THEN
			   fnLogMsg(ADR(LogMsg_0), LOG_INFO, 'Event is locked keep msg in Q Send Event ID %d,ErrorId =%d, flowid %d',
								AxisCtrlPtr^.Output.Error.ErrorEntry.MotorEvents  ,
								UDINT_TO_DINT(AxisCtrlPtr^.Output.Error.ErrorEntry.ErrorId),							
								AxisCtrlPtr^.Input.Parameter.pFlowID^);
			ELSE
				
			   fnLogMsg(ADR(LogMsg_0), LOG_INFO, 'Event is locked keep msg in Q Send Event ID %d,ErrorId =%d THERE IS NO LINK TO FLOW ID:',
								AxisCtrlPtr^.Output.Error.ErrorEntry.MotorEvents  ,
								UDINT_TO_DINT(AxisCtrlPtr^.Output.Error.ErrorEntry.ErrorId),							
								0);
			END_IF							
		ELSE

							
			IF AxisCtrlPtr^.Output.Error.ErrorEntry.ErrorId <>0 THEN
				
				LastErrorId := 	AxisCtrlPtr^.Output.Error.ErrorEntry.ErrorId;	
				
			END_IF
			
			PrevErrorId := AxisCtrlPtr^.Output.Error.ErrorEntry.ErrorId;
	
		END_IF
		
		lastEventID := 	AxisCtrlPtr^.Output.Error.ErrorEntry.MotorEvents;
		
	ELSIF MotorErrorQ.CheckQReadAvailable() THEN
					
	
			IF MotorErrorQ.ReadCurrentEntry(ADR(PrevMotorEvents),SIZEOF(Eh_ErrorEntry_typ)) THEN	
	
				IF Meth_GetEvent( PrevMotorEvents )  THEN
						
					MotorErrorQ.Dequeue(ADR(PrevMotorEvents),SIZEOF(PrevMotorEvents));
					
					fnLogMsg(ADR(LogMsg_0), LOG_INFO, 'Dequeue Event ID %d,ErrorId =%d',
								PrevMotorEvents.MotorEvents  ,
								UDINT_TO_DINT(PrevMotorEvents.ErrorId),							
								0);
	
				END_IF
			END_IF
	END_IF
	
END_IF
//fnLogTransfer FUNCTION call
fbPrgmBasic();

fnLogTransfer(ADR(LogMsg_0));

METHOD Meth_GetEvent : BOOL
VAR_INPUT
	ErrorEntry		: Eh_ErrorEntry_typ;
END_VAR
VAR
	EventSentOk:  	BOOL;
END_VAR
   EventSentOk := FALSE;

	CASE ErrorEntry.MotorEvents OF
		enumMotorEvents.NoEvents				:
			 EventSentOk := TRUE;//No Event	
		enumMotorEvents.MotorPositionError      :
			
			IF Meth_SendEvent( Ref_ev_MOTOR_POSITION ) = FALSE THEN
				EventSentOk := FALSE;
			ELSE
				EventSentOk := TRUE;
			END_IF
				
		enumMotorEvents.MotorSpeedError	        :
			IF Meth_SendEvent(  Ref_ev_MOTOR_Speed ) = FALSE THEN
				EventSentOk := FALSE;
			ELSE
				EventSentOk := TRUE;
			END_IF
		enumMotorEvents.MotorHomeNotFound	    :
			IF Meth_SendEvent( Ref_ev_HOME_NOT_FOUND ) = FALSE THEN
				EventSentOk := FALSE;
			ELSE
				EventSentOk := TRUE;
			END_IF
		enumMotorEvents.MotorOverCurrent	    :
			IF Meth_SendEvent( Ref_ev_OVER_CURRENT ) = FALSE THEN
				EventSentOk := FALSE;
			ELSE
				EventSentOk := TRUE;
			END_IF
		enumMotorEvents.MotorOverTemp		    :
			IF Meth_SendEvent(Ref_ev_MOTOR_OVER_TEMP ) = FALSE THEN
				EventSentOk := FALSE;
			ELSE
				EventSentOk := TRUE;
			END_IF
		enumMotorEvents.MotorFeedBackErr	    :
			IF Meth_SendEvent( Ref_ev_MOTOR_FEEDBACK_ERROR ) = FALSE THEN
				EventSentOk := FALSE;
			ELSE
				EventSentOk := TRUE;
			END_IF
		enumMotorEvents.MotorGeneralError		:
			IF Meth_SendEvent(Ref_ev_MOTOR_GENERAL_ERROR ) = FALSE THEN
				EventSentOk := FALSE;
			ELSE
				EventSentOk := TRUE;
			END_IF
		enumMotorEvents.MotorStalled			:
			IF Meth_SendEvent( Ref_ev_MOTOR_STALLED ) = FALSE THEN
				EventSentOk := FALSE;
			ELSE
				EventSentOk := TRUE;
			END_IF
		enumMotorEvents.MotorSupplyError		:
			IF Meth_SendEvent( Ref_ev_MOTOR_SUPPLY_ERROR ) = FALSE THEN
				EventSentOk := FALSE;
			ELSE
				EventSentOk := TRUE;
			END_IF
		enumMotorEvents.PLCillegalMsg			:
			IF Meth_SendEvent(Ref_ev_PLC_ILLEGAL_MSG ) = FALSE THEN
				EventSentOk := FALSE;
			ELSE
				EventSentOk := TRUE;
			END_IF
		enumMotorEvents.PLCIllegalParam			:
			IF Meth_SendEvent( Ref_ev_PLC_ILLEGAL_PARAM ) = FALSE THEN
				EventSentOk := FALSE;
			ELSE
				EventSentOk := TRUE;
			END_IF
		enumMotorEvents.DriveNotEnabled		    :
			IF Meth_SendEvent(Ref_ev_Drive_Not_Enabled ) = FALSE THEN
				EventSentOk := FALSE;
			ELSE
				EventSentOk := TRUE;
			END_IF
		enumMotorEvents.DriveNotReady           :
			IF Meth_SendEvent(Ref_ev_DRIVE_NOT_READY  ) = FALSE THEN
				EventSentOk := FALSE;
			ELSE
				EventSentOk := TRUE;
			END_IF
		enumMotorEvents.DriveComError           :
			IF Meth_SendEvent(Ref_ev_Drive_ComError ) = FALSE THEN
				EventSentOk := FALSE;
			ELSE
				EventSentOk := TRUE;
			END_IF
		enumMotorEvents.BreakResistorError:
			IF Meth_SendEvent( Ref_ev_BRAKE_RESISTOR_ERROR)= FALSE THEN
				EventSentOk := FALSE;
			ELSE
				EventSentOk := TRUE;
			END_IF
		
	END_CASE
	
		IF EventSentOk  AND ErrorEntry.MotorEvents <> enumMotorEvents.NoEvents THEN
			IF AxisCtrlPtr^.Input.Parameter.pFlowID <> 0 THEN
				fnLogMsg(ADR(LogMsg_0), LOG_INFO, 'Send Event ID %d,ErrorId =%d, FlowId=%d',
					AxisCtrlPtr^.Output.Error.ErrorEntry.MotorEvents  ,
					UDINT_TO_DINT(AxisCtrlPtr^.Output.Error.ErrorEntry.ErrorId),							
					AxisCtrlPtr^.Input.Parameter.pFlowID^);
			ELSE
				fnLogMsg(ADR(LogMsg_0), LOG_INFO, 'Send Event ID %d,ErrorId =%d, THERE IS NO LINK TO FLOWID',
					AxisCtrlPtr^.Output.Error.ErrorEntry.MotorEvents  ,
					UDINT_TO_DINT(AxisCtrlPtr^.Output.Error.ErrorEntry.ErrorId),							
					0);
		
			END_IF		
		END_IF

	Meth_GetEvent := EventSentOk;
END_METHOD

METHOD Meth_SendEvent : BOOL
VAR_INPUT
	RefEvent : REFERENCE TO EventHelper;
END_VAR
VAR

	Dummy :DINT :=0;
//	pFlowID :POINTER TO DINT;
END_VAR
IF __ISVALIDREF(RefEvent) THEN
		
		EventHeader.SubsysID :=			 AxisCtrlPtr^.Input.Parameter.SubsysID; 
		IF AxisCtrlPtr^.Input.Parameter.pFlowID <> 0 THEN
			EventHeader.pFlowID :=  AxisCtrlPtr^.Input.Parameter.pFlowID;					 // Flow ID
		ELSE
			EventHeader.pFlowID :=  ADR(Dummy);
		END_IF	
		EventParameters.MotorID := 		 AxisCtrlPtr^.Input.Parameter.MotorID; 	// Motor ID
		EventParameters.VendorNameID :=  AxisCtrlPtr^.Input.Parameter.Drive.VendorNameID;	// Vendor name ID

		fbPrgmBasic.mEventThrow(RefEvent,ADR(EventHeader),ADR(EventParameters) );			//RefEvent();
		Meth_SendEvent := TRUE;

END_IF
END_METHOD

END_FUNCTION_BLOCK

// ---- POUs/Lib/System/Queue.TcPOU

FUNCTION_BLOCK Queue EXTENDS FB_BaseFb
VAR_INPUT
	{attribute 'OPC.UA.DA' := '0'}
	busySem : BOOL :=FALSE; //used for test and set from outside call
END_VAR

VAR_OUTPUT
	
END_VAR
{attribute 'OPC.UA.DA' := '0'}
VAR CONSTANT
     QUEUE_SIZE  : UINT := 15;
END_VAR

VAR
	{attribute 'OPC.UA.DA' := '0'}
	StructSize : UDINT;
	{attribute 'OPC.UA.DA' := '0'}
	QArr	: ARRAY[0..QUEUE_SIZE] OF STRING[1000];	
	{attribute 'OPC.UA.DA' := '0'}
	pQArr  : POINTER TO  STRING;	
	{attribute 'OPC.UA.DA' := '0'}
	QWriteAdr :POINTER TO  STRING;
	{attribute 'OPC.UA.DA' := '0'}
	QReadAdr : POINTER TO  STRING;
	{attribute 'OPC.UA.DA' := '0'}
	pRead : UDINT;
	{attribute 'OPC.UA.DA' := '0'}
	pWrite :UDINT;
	{attribute 'OPC.UA.DA' := '0'}
	isInitDone :BOOL;
	{attribute 'OPC.UA.DA' := '0'}
	IsOverflow : BOOL;
	{attribute 'OPC.UA.DA' := '0'}
	isBusy :BOOL;	
	{attribute 'OPC.UA.DA' := '0'}
	isFull	: BOOL;
	{attribute 'OPC.UA.DA' := '0'}
	o_isEmpty : BOOL;
	{attribute 'OPC.UA.DA' := '0'}
	Error : BOOL;
	{attribute 'OPC.UA.DA' := '0'}
	ErrorID :USINT;
	{attribute 'OPC.UA.DA' := '0'}
	WriteMsgCount : UDINT;
	{attribute 'OPC.UA.DA' := '0'}
	ReadMsgCount  : UDINT;
	{attribute 'OPC.UA.DA' := '0'}
	o_EntriesCount : UINT;
	
END_VAR

METHOD CheckQReadAvailable : BOOL
VAR_INPUT
END_VAR

IF (isEmpty=FALSE) AND (isBusy = FALSE) THEN
	CheckQReadAvailable:= TRUE;
ELSE	
	CheckQReadAvailable:= FALSE;	
END_IF
END_METHOD

METHOD CheckQWriteAvailable : BOOL
VAR_INPUT
END_VAR

IF (isFull=FALSE) AND (isBusy = FALSE) THEN
	CheckQWriteAvailable:= TRUE;
	
ELSE
	
	CheckQWriteAvailable:= FALSE;	
END_IF
END_METHOD

METHOD Clear : BOOL
VAR_INPUT
END_VAR
		memset(pQArr,0,SIZEOF(QArr));
		pRead		:=0;
		pWrite		:=0;
		
		isInitDone 		:= TRUE;
		o_isEmpty		:=TRUE;
		isFull			:=FALSE;	
		isBusy			:=FALSE;
		Error			:=FALSE;
		ErrorID			:=0;
		
		o_EntriesCount := 0;
END_METHOD

METHOD Dequeue : BOOL
VAR_INPUT
	pReadData : POINTER TO BYTE;
	MsgLength  : UDINT;
END_VAR

IF THIS^.o_EntriesCount > 0 THEN	
	QReadAdr		:= (pQArr)+(pRead*StructSize);	
	memcpy(pReadData,QReadAdr,MsgLength);// (pDest,pSrc,length)
	THIS^.o_EntriesCount	:= THIS^.o_EntriesCount - 1;	
	pRead:=pRead+1;
	
	IF THIS^.pRead >= QUEUE_SIZE THEN
		THIS^.pRead	:= 0;
	END_IF	
	
    THIS^.IsFull		:= FALSE;
	ReadMsgCount:=ReadMsgCount+1;
	IF pRead=pWrite THEN
		o_isEmpty:=TRUE;
	END_IF	
		
END_IF
END_METHOD

METHOD Enqueue : BOOL
VAR_INPUT
	pWriteData : POINTER TO BYTE;	
	MsgLength  : UDINT;
END_VAR
IF o_EntriesCount < QUEUE_SIZE THEN
	isBusy := TRUE;
	QWriteAdr				:=(pQArr)+(pWrite*StructSize);
		IF MsgLength>0 AND (MsgLength<=StructSize)THEN
			memcpy(QWriteAdr,pWriteData,MsgLength);// (pDest,pSrc,length)  		
		ELSIF (MsgLength>StructSize)THEN
			Error		:=TRUE;
			ErrorID 	:= 5;
			memcpy(QWriteAdr,pWriteData,StructSize);// (pDest,pSrc,length)
		ELSE	// MsgLength = 0
			memcpy(QWriteAdr,pWriteData,StructSize);// (pDest,pSrc,length)	
		END_IF;
		pWrite:=pWrite+1;
		WriteMsgCount:=WriteMsgCount+1;
	// increase entries counter
	THIS^.o_EntriesCount	:= THIS^.o_EntriesCount + 1;	
		
	IF pWrite>=(QUEUE_SIZE) THEN
		pWrite:=0;
	END_IF;	
	
	THIS^.o_isEmpty		:= FALSE;
	IF THIS^.o_EntriesCount >= QUEUE_SIZE THEN
		THIS^.IsFull	:= TRUE;
	END_IF	
	
	IF WriteMsgCount>10000000 THEN
		WriteMsgCount:=0;
	END_IF;			
	isBusy := FALSE;
ELSE
	THIS^.IsOverflow	:= TRUE;	
END_IF
END_METHOD

PROPERTY EntriesCount : UINT
GET
EntriesCount :=o_EntriesCount;
END_GET
SET
END_SET
END_PROPERTY

METHOD FB_init : BOOL
VAR_INPUT
	bInitRetains : BOOL; // if TRUE, the retain variables are initialized (warm start / cold start)
	bInCopyCode : BOOL;  // if TRUE, the instance afterwards gets moved into the copy code (online change)
END_VAR
		THIS^.pQArr := ADR(QArr);		
		StructSize := SIZEOF(QArr[0]);
		
		memset(pQArr,0,SIZEOF(QArr));
		pRead		:=0;
		pWrite		:=0;
		
		isInitDone 		:= TRUE;
		o_isEmpty		:=TRUE;
		isFull			:=FALSE;	
		isBusy			:=FALSE;
		Error			:=FALSE;
		ErrorID			:=0;
		
		o_EntriesCount := 0;
END_METHOD

PROPERTY isEmpty : BOOL
GET
isEmpty := o_isEmpty;
END_GET
SET
END_SET
END_PROPERTY

METHOD Peek : BOOL
VAR_INPUT
END_VAR
END_METHOD

METHOD ReadCurrentEntry : BOOL//Only Read not Pop
VAR_INPUT
	pReadData : POINTER TO BYTE;
	MsgLength  : UDINT;
END_VAR

IF THIS^.o_EntriesCount > 0 THEN	
	QReadAdr		:= (pQArr)+(pRead*StructSize);	
	memcpy(pReadData,QReadAdr,MsgLength);// (pDest,pSrc,length)
	ReadCurrentEntry := TRUE;	
ELSE
	ReadCurrentEntry := FALSE;	
END_IF
END_METHOD

END_FUNCTION_BLOCK

// ---- POUs/Lib/System/FB_BaseFb.TcPOU
//
// In order for extender of this FB
// -- to set specific logger name category call SetLoggerCategoryName(<the name>) (from FB_Init())

FUNCTION_BLOCK FB_BaseFb
VAR
	{attribute 'OPC.UA.DA' := '0'}
	LogMsg_0: LogMsg;
	{attribute 'OPC.UA.DA' := '0'}
	pLogMsgToUse: POINTER TO LogMsg := ADR(LogMsg_0);
	{attribute 'OPC.UA.DA' := '0'}
	DINT_0 :DINT;
	
END_VAR

METHOD FB_init : BOOL
VAR_INPUT
	bInitRetains : BOOL; // if TRUE, the retain variables are initialized (warm start / cold start)
	bInCopyCode : BOOL;  // if TRUE, the instance afterwards gets moved into the copy code (online change)
END_VAR
END_METHOD

METHOD PUBLIC GetLoggerCategoryName : pointer to string
VAR_INPUT
END_VAR
GetLoggerCategoryName	:= ADR(THIS^.pLogMsgToUse^.logData.category);
END_METHOD

METHOD LogError
VAR_INPUT
	textMessage : STRING[LOG_MSG_TEXT_LENGTH];
	param1 : DINT;
	param2 : DINT;
	param3 : DINT;	
	param4 : DINT;
	param5 : DINT;
	param6 : DINT;	
END_VAR
pLogMsgToUse^.LogMsg(LOG_ERROR, textMessage, param1, param2, param3, param4, param5, param6);
LogTransfer();
END_METHOD

METHOD LogError_v2 : BOOL
VAR_INPUT
	textMessage : STRING[LOG_MSG_TEXT_LENGTH];
	param1 : ANY;
	param2 : ANY;
	param3 : ANY;	
	param4 : ANY;
	param5 : ANY;
	param6 : ANY;	
	param7 : ANY;	
	param8 : ANY;
	param9 : ANY;
	param10 : ANY;		
END_VAR
VAR
	param1_Arg   :T_arg;
	param2_Arg   :T_arg;
	param3_Arg   :T_arg;
	param4_Arg   :T_arg;
	param5_Arg   :T_arg;
	param6_Arg   :T_arg;
	param7_Arg   :T_arg;
	param8_Arg   :T_arg;
	param9_Arg   :T_arg;
	param10_Arg  :T_arg;
END_VAR

param1_Arg	:=fnCnvToTarg(param1);
param2_Arg	:=fnCnvToTarg(param2);
param3_Arg	:=fnCnvToTarg(param3);
param4_Arg	:=fnCnvToTarg(param4);
param5_Arg	:=fnCnvToTarg(param5);
param6_Arg	:=fnCnvToTarg(param6);
param7_Arg	:=fnCnvToTarg(param7);
param8_Arg	:=fnCnvToTarg(param8);
param9_Arg	:=fnCnvToTarg(param9);
param10_Arg	:=fnCnvToTarg(param10);

pLogMsgToUse^.LogMsg_v2(LOG_ERROR, textMessage, param1_Arg, param2_Arg, param3_Arg, param4_Arg, param5_Arg, param6_Arg, param7_Arg ,param8_Arg ,param9_Arg,param10_Arg);
LogTransfer();
END_METHOD

METHOD LogInfo
VAR_INPUT
	textMessage : STRING[LOG_MSG_TEXT_LENGTH];
	param1 : DINT;
	param2 : DINT;
	param3 : DINT;	
	param4 : DINT;
	param5 : DINT;
	param6 : DINT;	
END_VAR
pLogMsgToUse^.LogMsg(LOG_INFO, textMessage, param1, param2, param3, param4, param5, param6);
LogTransfer();
END_METHOD

METHOD LogInfo_v2 : BOOL
VAR_INPUT
	textMessage : STRING[LOG_MSG_TEXT_LENGTH];
	param1 : ANY;
	param2 : ANY;
	param3 : ANY;	
	param4 : ANY;
	param5 : ANY;
	param6 : ANY;	
	param7 : ANY;	
	param8 : ANY;
	param9 : ANY;
	param10 : ANY;		
END_VAR
VAR
	param1_Arg   :T_arg;
	param2_Arg   :T_arg;
	param3_Arg   :T_arg;
	param4_Arg   :T_arg;
	param5_Arg   :T_arg;
	param6_Arg   :T_arg;
	param7_Arg   :T_arg;
	param8_Arg   :T_arg;
	param9_Arg   :T_arg;
	param10_Arg  :T_arg;
END_VAR

param1_Arg	:=fnCnvToTarg(param1);
param2_Arg	:=fnCnvToTarg(param2);
param3_Arg	:=fnCnvToTarg(param3);
param4_Arg	:=fnCnvToTarg(param4);
param5_Arg	:=fnCnvToTarg(param5);
param6_Arg	:=fnCnvToTarg(param6);
param7_Arg	:=fnCnvToTarg(param7);
param8_Arg	:=fnCnvToTarg(param8);
param9_Arg	:=fnCnvToTarg(param9);
param10_Arg	:=fnCnvToTarg(param10);

pLogMsgToUse^.LogMsg_v2(LOG_INFO, textMessage, param1_Arg, param2_Arg, param3_Arg, param4_Arg, param5_Arg, param6_Arg, param7_Arg ,param8_Arg ,param9_Arg,param10_Arg);
LogTransfer();
END_METHOD

METHOD LogTransfer
fnLogTransfer(pLogMsgToUse);
END_METHOD

METHOD LogWarning
VAR_INPUT
	textMessage : STRING[LOG_MSG_TEXT_LENGTH];
	param1 : DINT;
	param2 : DINT;
	param3 : DINT;	
	param4 : DINT;
	param5 : DINT;
	param6 : DINT;	
END_VAR
pLogMsgToUse^.LogMsg(LOG_WARNING, textMessage, param1, param2, param3, param4, param5, param6);
LogTransfer();
END_METHOD

METHOD LogWarning_v2 : BOOL
VAR_INPUT
	textMessage : STRING[LOG_MSG_TEXT_LENGTH];
	param1 : ANY;
	param2 : ANY;
	param3 : ANY;	
	param4 : ANY;
	param5 : ANY;
	param6 : ANY;	
	param7 : ANY;	
	param8 : ANY;
	param9 : ANY;
	param10 : ANY;		
END_VAR
VAR
	param1_Arg   :T_arg;
	param2_Arg   :T_arg;
	param3_Arg   :T_arg;
	param4_Arg   :T_arg;
	param5_Arg   :T_arg;
	param6_Arg   :T_arg;
	param7_Arg   :T_arg;
	param8_Arg   :T_arg;
	param9_Arg   :T_arg;
	param10_Arg  :T_arg;
END_VAR

param1_Arg	:=fnCnvToTarg(param1);
param2_Arg	:=fnCnvToTarg(param2);
param3_Arg	:=fnCnvToTarg(param3);
param4_Arg	:=fnCnvToTarg(param4);
param5_Arg	:=fnCnvToTarg(param5);
param6_Arg	:=fnCnvToTarg(param6);
param7_Arg	:=fnCnvToTarg(param7);
param8_Arg	:=fnCnvToTarg(param8);
param9_Arg	:=fnCnvToTarg(param9);
param10_Arg	:=fnCnvToTarg(param10);

pLogMsgToUse^.LogMsg_v2(LOG_WARNING, textMessage, param1_Arg, param2_Arg, param3_Arg, param4_Arg, param5_Arg, param6_Arg, param7_Arg ,param8_Arg ,param9_Arg,param10_Arg);
LogTransfer();
END_METHOD

METHOD SetLogger
VAR_INPUT
	logMsgToUse: REFERENCE TO LogMsg;
END_VAR
IF(__ISVALIDREF(logMsgToUse)) THEN
	pLogMsgToUse := ADR(logMsgToUse);
END_IF
END_METHOD

METHOD SetLoggerCategoryName
VAR_INPUT
	categoryName: STRING;	// Removed "REFERENCE TO "
END_VAR
categoryName[LOG_MSG_CATEGORY_LENGTH - 1] := 0;

// do not use pLogMsgToUse since the external logger logger could has be set
LogMsg_0.InitLogger(categoryName, 0,0);
END_METHOD

END_FUNCTION_BLOCK

// ---- POUs/Lib/System/fnCnvToTarg.TcPOU
FUNCTION fnCnvToTarg : T_Arg
VAR_INPUT
	param1:ANY;
END_VAR
VAR
END_VAR


CASE 	 param1.TypeClass OF	
	 __SYSTEM.TYPE_CLASS.TYPE_REAL:
			 fnCnvToTarg.eType	:= E_ArgType.ARGTYPE_REAL;
	 __SYSTEM.TYPE_CLASS.TYPE_INT:
			 fnCnvToTarg.eType	:= E_ArgType.ARGTYPE_INT;	 
	 __SYSTEM.TYPE_CLASS.TYPE_LREAL:
			 fnCnvToTarg.eType	:= E_ArgType.ARGTYPE_LREAL;
	 __SYSTEM.TYPE_CLASS.TYPE_SINT:
			 fnCnvToTarg.eType	:= E_ArgType.ARGTYPE_SINT;	 		
	 __SYSTEM.TYPE_CLASS.TYPE_DINT:
			 fnCnvToTarg.eType	:= E_ArgType.ARGTYPE_DINT;
	 __SYSTEM.TYPE_CLASS.TYPE_USINT:
			 fnCnvToTarg.eType	:= E_ArgType.ARGTYPE_USINT;	 
	 __SYSTEM.TYPE_CLASS.TYPE_UINT:
			 fnCnvToTarg.eType	:= E_ArgType.ARGTYPE_UINT;
	 __SYSTEM.TYPE_CLASS.TYPE_UDINT:
			 fnCnvToTarg.eType	:= E_ArgType.ARGTYPE_UDINT;	 	
	 __SYSTEM.TYPE_CLASS.TYPE_ULINT:
			 fnCnvToTarg.eType	:= E_ArgType.ARGTYPE_ULARGE;
	__SYSTEM.TYPE_CLASS.TYPE_LINT:
			 fnCnvToTarg.eType	:= E_ArgType.ARGTYPE_LARGE;	 			 
	 __SYSTEM.TYPE_CLASS.TYPE_STRING:
			 fnCnvToTarg.eType	:= E_ArgType.ARGTYPE_STRING;
	 __SYSTEM.TYPE_CLASS.TYPE_BOOL:
			 fnCnvToTarg.eType	:= E_ArgType.ARGTYPE_BYTE;//Not a Bug use to convert bool to byte for string format	 
	 __SYSTEM.TYPE_CLASS.TYPE_BYTE:
			 fnCnvToTarg.eType	:= E_ArgType.ARGTYPE_BYTE;
	 __SYSTEM.TYPE_CLASS.TYPE_WORD:
			 fnCnvToTarg.eType	:= E_ArgType.ARGTYPE_WORD;	 		
	 __SYSTEM.TYPE_CLASS.TYPE_DWORD:
			 fnCnvToTarg.eType	:= E_ArgType.ARGTYPE_DWORD;
	 __SYSTEM.TYPE_CLASS.TYPE_ENUM:
	 		IF param1.diSize = SIZEOF(INT) THEN
			 	fnCnvToTarg.eType	:= E_ArgType.ARGTYPE_INT;	
			ELSIF param1.diSize = SIZEOF(DINT) THEN		 
				fnCnvToTarg.eType	:= E_ArgType.ARGTYPE_DINT;	
			ELSIF param1.diSize = SIZEOF(UDINT) THEN		 
				fnCnvToTarg.eType	:= E_ArgType.ARGTYPE_UDINT;			
			ELSIF param1.diSize = SIZEOF(UINT) THEN		 
				fnCnvToTarg.eType	:= E_ArgType.ARGTYPE_UINT;	
			END_IF	
ELSE
	RETURN; 
END_CASE

fnCnvToTarg.pData := param1.pValue;
fnCnvToTarg.cbLen := DINT_TO_UDINT(param1.diSize);

END_FUNCTION

// ---- POUs/Lib/ProgramBasic/FB_PrgmBasic.TcPOU
FUNCTION_BLOCK FB_PrgmBasic
VAR_INPUT
	
	EventParameters:	EventParam_Typ;	
	EventHeader:		EventHeader_Typ;	
END_VAR
VAR_OUTPUT
END_VAR
VAR
	LocalEventQ	: Queue;
	LocalEventObj :LocalEvent_Typ;
	GlobalEventObj :LocalEvent_Typ;
	FlagSendEvent :BOOL;
	FlagActive	:BOOL;
	DummyFlowID: DINT := 0;
END_VAR

//Check if Q has elements
IF THIS^.LocalEventQ.EntriesCount >0 AND (FlagSendEvent=FALSE)  THEN
	THIS^.LocalEventQ.Dequeue(ADR(THIS^.GlobalEventObj),SIZEOF(LocalEvent_Typ));
	FlagSendEvent:=TRUE;
END_IF


IF FlagSendEvent THEN
	IF TestAndSet(THIS^.GlobalEventObj.rEvent.Busy) THEN // Check if the event FB is free
		FlagActive:=TRUE;	
	END_IF
	IF FlagActive THEN
//		THIS^.GlobalEventObj.rEvent(pFlowID:=ADR(GlobalEventObj.flowId),pEvPar:=ADR(GlobalEventObj.EventParameters)); //Call the event FB 
		THIS^.GlobalEventObj.rEvent(pEvHeader:=ADR(GlobalEventObj.EventHeader),pEvPar:=ADR(GlobalEventObj.EventParameters)); //Call the event FB 
		IF THIS^.GlobalEventObj.rEvent.Done THEN
			THIS^.GlobalEventObj.rEvent.Done 	:=FALSE;
			THIS^.GlobalEventObj.rEvent.Busy	:=FALSE;//Free FB
			FlagActive:=FALSE;
			FlagSendEvent:=FALSE;
		END_IF
	END_IF
END_IF

METHOD mEventThrow : BOOL
VAR_INPUT
	rEvent : REFERENCE TO EventHelper;
//	pFlowID :POINTER TO DINT;
	pEvHeader: POINTER TO EventHeader_Typ;
	pEvPar: POINTER TO EventParam_Typ;


END_VAR
IF (pEvHeader^.pFlowID = 0) THEN
	pEvHeader^.pFlowID := ADR(DummyFlowID);
END_IF
//Dereference data
LocalEventObj.EventParameters := pEvPar^;
LocalEventObj.rEvent REF= rEvent;
//LocalEventObj.flowId := pFlowID^;
LocalEventObj.EventHeader := pEvHeader^;
	
LocalEventQ.Enqueue(ADR(THIS^.LocalEventObj),SIZEOF(THIS^.LocalEventObj));
mEventThrow:=TRUE;
END_METHOD

END_FUNCTION_BLOCK

// ---- POUs/Lib/Events/EventHelper.TcPOU

FUNCTION_BLOCK EventHelper EXTENDS FB_BaseFb
VAR_INPUT
//	pFlowID: 	POINTER TO DINT;
	pEvHeader: 	POINTER TO EventHeader_Typ;
	pEvPar: 	POINTER TO EventParam_Typ;
	Busy:BOOL:=FALSE;
	Done:BOOL;
END_VAR
VAR_OUTPUT
	
END_VAR
VAR
	EventReport :EventReport_Typ;
	InitDone:	 BOOL;
END_VAR

IF NOT InitDone THEN
	mInit();
	InitDone:= TRUE;
END_IF

METHOD mInit : BOOL
VAR_INPUT
END_VAR
SetLoggerCategoryName('Events');
END_METHOD

END_FUNCTION_BLOCK

// ---- POUs/Lib/Events/Demo/DemoProgram.TcPOU
PROGRAM DemoProgram
VAR
	{attribute 'OPC.UA.DA' := '1'}
    //{attribute 'OPC.UA.DA.StructuredType' := '1'}
//	Events:EventsFB;
	
	fbProgramBase :FB_PrgmBasic;
	//EventParameters:EventParam_Typ;	
	flowid:DINT;
	testevent:BOOL;
	refEvent :REFERENCE TO EventHelper;
END_VAR


//EventParameters.par2:=2;
IF testevent THEN
	fbProgramBase.EventParameters.Par1:=1;
//	fbProgramBase.mEventThrow(ev_PLC_ILLEGAL_MSG,ADR(flowid),ADR(fbProgramBase.EventParameters));
	fbProgramBase.mEventThrow(ev_PLC_ILLEGAL_MSG,ADR(fbProgramBase.EventHeader),ADR(fbProgramBase.EventParameters));
	
	fbProgramBase.EventParameters.Par1:=3;
//	fbProgramBase.mEventThrow(ev_PLC_INTERNAL_TIMEOUT,ADR(flowid),ADR(fbProgramBase.EventParameters));
	fbProgramBase.mEventThrow(ev_PLC_INTERNAL_TIMEOUT,ADR(fbProgramBase.EventHeader),ADR(fbProgramBase.EventParameters));

		fbProgramBase.EventParameters.Par1:=5;
//	fbProgramBase.mEventThrow(ev_PLC_ILLEGAL_MSG,ADR(flowid),ADR(fbProgramBase.EventParameters));
	fbProgramBase.mEventThrow(ev_PLC_ILLEGAL_MSG,ADR(fbProgramBase.EventHeader),ADR(fbProgramBase.EventParameters));
	
		fbProgramBase.EventParameters.Par1:=3;
//	fbProgramBase.mEventThrow(ev_PLC_INTERNAL_TIMEOUT,ADR(flowid),ADR(fbProgramBase.EventParameters));
	fbProgramBase.mEventThrow(ev_PLC_INTERNAL_TIMEOUT,ADR(fbProgramBase.EventHeader),ADR(fbProgramBase.EventParameters));
	testevent:=FALSE;
END_IF


fbProgramBase();

END_PROGRAM

// ---- POUs/Lib/Events/EventQueue.TcPOU
FUNCTION_BLOCK EventQueue EXTENDS Queue
VAR_INPUT
END_VAR
VAR_OUTPUT
	{attribute 'OPC.UA.DA' := '1'}
    {attribute 'OPC.UA.DA.StructuredType' := '1'}
	ErrorEvent:EventReport_Typ;		
END_VAR
VAR
	{attribute 'OPC.UA.DA' := '0'}
	EventActiveFlag:BOOL;
	{attribute 'OPC.UA.DA' := '0'}
	InitDone:		BOOL;
	{attribute 'OPC.UA.DA' := '0'}
    SubsystemIDString:	STRING;

END_VAR
VAR_STAT
	{attribute 'OPC.UA.DA' := '0'}
	SequentialID:	DINT;
END_VAR

IF NOT InitDone THEN
	mInit();
	InitDone:= TRUE;
END_IF
IF THIS^.EntriesCount > 0 AND (THIS^.CheckQReadAvailable()) AND EventActiveFlag=FALSE  THEN
	EventActiveFlag:=TRUE;
    THIS^.Dequeue(ADR(ErrorEvent),SIZEOF(ErrorEvent));
	SequentialID := SequentialID + 1 ;
	IF SequentialID >= 16#7FFFFFFF THEN
		SequentialID := 0;
	END_IF

	ErrorEvent.SequentialID := SequentialID;
	SubsystemIDString := TO_STRING(ErrorEvent.SubsysID);
	LogError_v2('Send event %s from %s, FlowID %d, SequentialID %d ' ,
		ErrorEvent.EventID, SubsystemIDString, ErrorEvent.FlowID,SequentialID,dint_0,dint_0,dint_0,dint_0,dint_0,dint_0);
END_IF

{attribute 'TcRpcEnable':='1'}
METHOD mAckEvent : BOOL
VAR_INPUT
END_VAR
EventActiveFlag:=FALSE;
MEMSET(ADR(ErrorEvent),0,SIZEOF(ErrorEvent));

mAckEvent := TRUE;
END_METHOD

{attribute 'TcRpcEnable':='1'}
METHOD mClearQueue : BOOL
VAR_INPUT
END_VAR
 THIS^.Clear();
 LogError_v2('Clear EventQueue ' ,dint_0, dint_0, dint_0,dint_0,dint_0,dint_0,dint_0,dint_0,dint_0,dint_0);
END_METHOD

METHOD mInit : BOOL
VAR_INPUT
END_VAR
SetLoggerCategoryName('Events');
END_METHOD

END_FUNCTION_BLOCK

// ---- POUs/Lib/IO/fb_IO_Basic.TcPOU
FUNCTION_BLOCK fb_IO_Basic
VAR_INPUT
END_VAR
VAR_OUTPUT
END_VAR
VAR
END_VAR

END_FUNCTION_BLOCK

// ---- POUs/Lib/IO/fb_io_in_bool.TcPOU
FUNCTION_BLOCK fb_io_in_bool
VAR_INPUT
	hw_value AT %I* 	: BOOL;
	SimFlag:BOOL;
	SimValue:BOOL:=TRUE;
END_VAR
VAR_OUTPUT
	Value:BOOL;
END_VAR
VAR
END_VAR


IF SimFlag THEN
	Value:= SimValue;
ELSE
	value:= hw_value;
END_IF

END_FUNCTION_BLOCK

// ---- POUs/Lib/Logging/HpString/AMSNETID_TO_STRING.TcPOU
FUNCTION AMSNETID_TO_STRING : STRING
VAR_INPUT
	AoeNetId 	: AMSNETID;
END_VAR
VAR
	Index		: INT := 0;
END_VAR

AMSNETID_TO_STRING := TO_STRING(AoeNetId[Index]);
FOR Index := 1 TO 5 DO
	AMSNETID_TO_STRING := CONCAT(AMSNETID_TO_STRING, '.');
	AMSNETID_TO_STRING := CONCAT(AMSNETID_TO_STRING, TO_STRING(AoeNetId[Index]));
END_FOR

END_FUNCTION

// ---- POUs/Lib/Logging/HpString/F_ADStoStr.TcPOU
FUNCTION F_ADStoStr :  STRING
VAR_INPUT
	ErrCode:    DWORD;
END_VAR
VAR
END_VAR

CASE ErrCode OF
	
	  0:    F_ADStoStr:=	'NoError ';		
      1:    F_ADStoStr:='InternalError ';
      2:    F_ADStoStr:='NoRTime ';
      3:    F_ADStoStr:='LockedMemoryError';
      4:    F_ADStoStr:='MailBoxError ';
      5:    F_ADStoStr:='WrongHMsg ';
      6:    F_ADStoStr:='TargetPortNotFound ';
      7:    F_ADStoStr:='TargetMachineNotFound ';
      8:    F_ADStoStr:='UnknownCommandID ';
      9:    F_ADStoStr:='BadTaskID ';
      10:   F_ADStoStr:= 'NoIO ';
      11:   F_ADStoStr:= 'UnknwonAmsCommand ';
      12:   F_ADStoStr:= 'Win32Error ';
      13:   F_ADStoStr:= 'PortNotConnected ';
      14:   F_ADStoStr:='InvalidAmsLength ';
      15:   F_ADStoStr:= 'InvalidAmsNetID ';
      16:   F_ADStoStr:= 'LowInstallLevel ';
      17:   F_ADStoStr:= 'NoDebug ';
      18:   F_ADStoStr:= 'PortDisabled ';
      19:   F_ADStoStr:= 'PortConnected ';
      20:   F_ADStoStr:= 'AmsSyncWin32Error ';
      21:   F_ADStoStr:= 'SyncTimeOut ';
      22:   F_ADStoStr:= 'AmsSyncAmsError ';
      23:   F_ADStoStr:= 'AmsSyncNoIndexMap ';
      24:   F_ADStoStr:= 'InvalidAmsPort ';
      25:   F_ADStoStr:= 'NoMemory ';
      26:    F_ADStoStr:= 'TCPSendError ';
      27:    F_ADStoStr:= 'HostUnreachable ';
      1280:  F_ADStoStr:=   'NoLockedMemory ';
      1282:  F_ADStoStr:=  'MailboxFull ';
      1792:  F_ADStoStr:=  'DeviceError ';
      1793:  F_ADStoStr:=  'DeviceServiceNotSupported ';
      1794:  F_ADStoStr:=  'DeviceInvalidGroup ';
      1795:  F_ADStoStr:=  'DeviceInvalidOffset ';
      1796:  F_ADStoStr:=  'DeviceInvalidAccess ';
      1797:  F_ADStoStr:=  'DeviceInvalidSize ';
      1798:  F_ADStoStr:=  'DeviceInvalidData ';
      1799:  F_ADStoStr:=  'DeviceNotReady ';
      1800:  F_ADStoStr:=  'DeviceBusy ';
      1801:  F_ADStoStr:=  'DeviceInvalidContext';
      1802:  F_ADStoStr:=  'DeviceNoMemory ';
      1803:  F_ADStoStr:=  'DeviceInavlidParam ';
      1804:  F_ADStoStr:=  'DeviceNotFound ';
      1805:  F_ADStoStr:=  'DeviceSyntaxError ';
      1806:  F_ADStoStr:= 'DeviceIncompatible ';
      1808:  F_ADStoStr:= 'DeviceSymbolNotFound ';
      1809:  F_ADStoStr:= 'DeviceSymbolVersionInvalid ';
      1810:  F_ADStoStr:=  'DeviceInvalidState ';
      1811:  F_ADStoStr:= 'DeviceTransModeNotSupported ';
      1812:  F_ADStoStr:= 'DeviceNotifyHandleInvalid ';
      1813:  F_ADStoStr:=  'DeviceClientUnknown ';
      1814:  F_ADStoStr:=  'DeviceNoMoreHandles ';
      1815:  F_ADStoStr:=  'DeviceInvalidWatchsize ';
      1816:  F_ADStoStr:=  'DeviceNotInitialized ';
      1817:  F_ADStoStr:=  'DeviceTimeOut ';
      1818:  F_ADStoStr:=  'DeviceNoInterface ';
      1819:  F_ADStoStr:= 'DeviceInvalidInterface ';
      1820:  F_ADStoStr:=  'DeviceInvalidCLSID ';
      1821:  F_ADStoStr:=  'DeviceInvalidObjectID ';
      1856:  F_ADStoStr:=  'ClientError ';
      1857:  F_ADStoStr:=  'ClientInvalidParameter ';
      1858:  F_ADStoStr:=  'ClientListEmpty ';
      1859:  F_ADStoStr:=  'ClientVaraiableInUse ';
      1860:  F_ADStoStr:=  'ClientDuplicateInvokeID ';
      1861:  F_ADStoStr:=  'ClientSyncTimeOut ';
      1862:  F_ADStoStr:=  'ClientW32OR ';
      1863:  F_ADStoStr:=  'ClientTimeoutInvalid ';
      1864:  F_ADStoStr:=  'ClientPortNotOpen ';
      1865:  F_ADStoStr:=  'ClientNoAmsAddr ';
      1872:  F_ADStoStr:=  'ClientSyncInternal ';
      1873:  F_ADStoStr:=  'ClientAddHash ';
      1874:  F_ADStoStr:=  'ClientRemoveHash ';
      1875:  F_ADStoStr:= 'ClientNoMoreSymbols ';
      1876:  F_ADStoStr:=  'ClientSyncResInvalid ';    
      1877:  F_ADStoStr:=  'ClientSyncPortLocked ';    
      32768: F_ADStoStr:=   'ClientQueueFull ';   

END_CASE

END_FUNCTION

// ---- POUs/Lib/Logging/logLib/fnLogMsg6.TcPOU
FUNCTION fnLogMsg6 : BOOL
VAR_INPUT
		logMsgPtr : POINTER TO LogMsg;
		messageLevel : enumLogMessageLevelSeverity;
		textMessage : STRING[LOG_MSG_TEXT_LENGTH];
		param1 : DINT;
		param2 : DINT;
		param3 : DINT;
		param4 : DINT;
		param5 : DINT;
		param6 : DINT;
END_VAR

fnLogMsg6 := logMsgPtr^.LogMsg(messageLevel, textMessage, param1, param2, param3, param4, param5, param6);

END_FUNCTION

// ---- POUs/Lib/Logging/logLib/fnLogStatusToString.TcPOU
FUNCTION fnLogStatusToString : STRING
VAR_INPUT
	
	eStatusType:	E_LogStatusReport_Type;
	LogData:		INT;
END_VAR
VAR		
	
END_VAR

IF eStatusType = E_LogStatusReport_Type.General THEN
	CASE LogData OF 
		E_SubSystemGeneralStatus.CommInit:
			fnLogStatusToString:=	'General - CommInit = 0';
		E_SubSystemGeneralStatus.PowerDisabled: 
			fnLogStatusToString:=	'General - PowerDisabled = 1';	
		E_SubSystemGeneralStatus.Off_DeEnergized:
			fnLogStatusToString:=	'General - Off_DeEnergized = 2';		 	
		E_SubSystemGeneralStatus.MechinitPassed: 
			fnLogStatusToString:=	'General - MechinitPassed = 3';			
		E_SubSystemGeneralStatus.Ready: 
			fnLogStatusToString:=	'General - Ready = 4';	
		E_SubSystemGeneralStatus.Printing: 
			fnLogStatusToString:=	'General - Printing = 5';		
		E_SubSystemGeneralStatus.FaultDisabled: 
			fnLogStatusToString:=	'General - FaultDisabled = 80';				
		E_SubSystemGeneralStatus.BusyStateTransition:  
			fnLogStatusToString:=	'General - BusyStateTransition = 90';
		E_SubSystemGeneralStatus.NotActive:  
			fnLogStatusToString:=	'General - BusyStateTransition = 100';
	END_CASE
	
ELSIF eStatusType = E_LogStatusReport_Type.Speed THEN	
	CASE LogData OF 
		E_SpeedStatus.IDLER:
			fnLogStatusToString:=	'Speed - NO_POWER_IDLER = 0';				
		E_SpeedStatus.STANDSTILL: 
			fnLogStatusToString:=	'Speed - STANDSTILL_SPEED_STATUS = 1';		
		E_SpeedStatus.AT_SPEED:	
			fnLogStatusToString:=	'Speed - AT_SPEED = 2';
		E_SpeedStatus.SYNCED_TO_MASTER :	
			fnLogStatusToString:=	'Speed - SYNCED_TO_MASTER = 3';
	END_CASE

ELSIF eStatusType = E_LogStatusReport_Type.Eng THEN	
	CASE LogData OF 		
		E_SubSysEngTarget.NoCMD:
			fnLogStatusToString:=	'Engage - NoCMD = 0';				
		E_SubSysEngTarget.DISENGAGE: 
			fnLogStatusToString:=	'Engage - DISENGAGE = 1';		
		E_SubSysEngTarget.ENGAGE:
			fnLogStatusToString:=	'Engage - ENGAGE = 2';
		E_SubSysEngTarget.SEMI_ENG:
			fnLogStatusToString:=	'Engage - SEMI_ENG = 3';
		
	END_CASE
ELSIF eStatusType = E_LogStatusReport_Type.EFS THEN	
	CASE LogData OF 
		E_Subsystem_EFS_Status.INACTIVE:
			fnLogStatusToString:=	'EFS - INACTIVE = 0';
		E_Subsystem_EFS_Status.PRE_CLEAN_ACTIVE:
			fnLogStatusToString:=	'EFS - PRE_CLEAN_ACTIVE = 1';
		E_Subsystem_EFS_Status.CLEAN_ACTIVE:
			fnLogStatusToString:=	'EFS - CLEAN_ACTIVE = 2';
 	END_CASE
				
END_IF

END_FUNCTION

// ---- POUs/Lib/Logging/PackData/getUsint.TcPOU
FUNCTION getUsint : BOOL
VAR_INPUT
END_VAR
VAR
END_VAR
VAR_IN_OUT
	usintRef : USINT;
	bufferRef : UDINT;
END_VAR

	memcpy(ADR(usintRef), bufferRef, SIZEOF(USINT));
	bufferRef := bufferRef + SIZEOF(USINT);
	getUsint := TRUE;

END_FUNCTION

// ---- POUs/Lib/Motion/CanOpenAxis/BeckHoff/BeckHoff8xxxAxis_FB.TcPOU
FUNCTION_BLOCK PUBLIC BeckHoff8xxxAxis_FB EXTENDS BeckHoffBasicAxis_FB  
VAR_INPUT		
	io_SafetyState: 	BYTE;	
END_VAR
VAR_IN_OUT	
END_VAR
VAR_OUTPUT	
END_VAR

VAR
//	DebugError					: UINT;
	Drive8000InitDone :BOOL := FALSE;
END_VAR

IF NOT Drive8000InitDone THEN
	Meth_Init();
	Drive8000InitDone := TRUE;
END_IF

AxisCtrlPtr^.Input.Parameter.Drive.eDriveType := enumDriveType.e8xxxBeckhoff;	
AxisCtrlPtr^.Input.Parameter.Drive.VendorNameID := eVendorNameID.Beckhoff;

SUPER^(AxisRef:=AxisRef);

AxisCtrlPtr^.Output.Status.DriveEnable:=	BYTE_TO_BOOL(io_SafetyState);

METHOD CreateDriveErrMsgDetails : enumMotorEvents
VAR_INPUT
	ErrorId			: UDINT;
END_VAR
CASE ErrorId OF
	
	16#0:
		CreateDriveErrMsgDetails := enumMotorEvents.NoEvents;
		fnLogMsg(ADR(LogMsg_0),LOG_ERROR,'Beckhoff Drive8 ErrorId %d  ,No error',UDINT_TO_DINT(ErrorId),0,0);
	16#2340: 
		CreateDriveErrMsgDetails := enumMotorEvents.MotorSupplyError ;
		fnLogMsg(ADR(LogMsg_0),LOG_ERROR,'Beckhoff Drive8 ErrorId %d  Short circuit (motor-side)',UDINT_TO_DINT(ErrorId),0,0);
	16#2380:
		CreateDriveErrMsgDetails := enumMotorEvents.MotorOverCurrent ;
		fnLogMsg(ADR(LogMsg_0),LOG_ERROR,'Beckhoff Drive8 ErrorId %d Continuous over current -U',UDINT_TO_DINT(ErrorId),0,0);
	16#2381:
		CreateDriveErrMsgDetails := enumMotorEvents.MotorOverCurrent ;
		fnLogMsg(ADR(LogMsg_0),LOG_ERROR,'Beckhoff Drive8 ErrorId %d Continuous over current - V',UDINT_TO_DINT(ErrorId),0,0);
	16#2382:
		CreateDriveErrMsgDetails := enumMotorEvents.MotorOverCurrent ;	
		fnLogMsg(ADR(LogMsg_0),LOG_ERROR,'Beckhoff Drive8 ErrorId %d Continuous over current Ohase W',UDINT_TO_DINT(ErrorId),0,0);
		
	16#2383:
		CreateDriveErrMsgDetails := enumMotorEvents.MotorSupplyError;
		fnLogMsg(ADR(LogMsg_0),LOG_ERROR,'Beckhoff Drive8 ErrorId %d Phase U current offset out of range',UDINT_TO_DINT(ErrorId),0,0);
	16#2384:
		CreateDriveErrMsgDetails := enumMotorEvents.MotorSupplyError;
		fnLogMsg(ADR(LogMsg_0),LOG_ERROR,'Beckhoff Drive8 ErrorId %d  Phase V current offset out of range',UDINT_TO_DINT(ErrorId),0,0);
	16#2385:
		CreateDriveErrMsgDetails := enumMotorEvents.MotorSupplyError;
		fnLogMsg(ADR(LogMsg_0),LOG_ERROR,'Beckhoff Drive8 ErrorId %d  Phase W current offset out of range',UDINT_TO_DINT(ErrorId),0,0);
	16#3180..16#3181 :
		CreateDriveErrMsgDetails := enumMotorEvents.MotorGeneralError;
		fnLogMsg(ADR(LogMsg_0),LOG_ERROR,'Beckhoff Drive8 ErrorId %d  Phase failure motor',UDINT_TO_DINT(ErrorId),0,0);
	16#3210: 
		CreateDriveErrMsgDetails := enumMotorEvents.MotorSupplyError;
		fnLogMsg(ADR(LogMsg_0),LOG_ERROR,'Beckhoff Drive ErrorId %d DC link overvoltage',UDINT_TO_DINT(ErrorId),0,0);
		
		
	16#3220:
		CreateDriveErrMsgDetails := enumMotorEvents.MotorSupplyError;
		fnLogMsg(ADR(LogMsg_0),LOG_ERROR,'Beckhoff Drive8 ErrorId %d DC-Link undervoltage',UDINT_TO_DINT(ErrorId),0,0);
	16#3280:
 		CreateDriveErrMsgDetails := enumMotorEvents.MotorSupplyError;
		fnLogMsg(ADR(LogMsg_0),LOG_ERROR,'Beckhoff Drive8 ErrorId %d 2  DC link is not ready',UDINT_TO_DINT(ErrorId),0,0);
	16#4310: 
		CreateDriveErrMsgDetails := enumMotorEvents.MotorOverTemp;
		fnLogMsg(ADR(LogMsg_0),LOG_ERROR,'Beckhoff Drive8 ErrorId %d Drive overtemperature ',UDINT_TO_DINT(ErrorId),0,0);
	16#4380:
		CreateDriveErrMsgDetails := enumMotorEvents.MotorOverTemp;
		fnLogMsg(ADR(LogMsg_0),LOG_ERROR,'Beckhoff Drive8 ErrorId %d  Fan speed seems to be zero',UDINT_TO_DINT(ErrorId),0,0);
	16#5112:
		CreateDriveErrMsgDetails := enumMotorEvents.MotorSupplyError;
		fnLogMsg(ADR(LogMsg_0),LOG_ERROR,'Beckhoff Drive8 ErrorId %d  Supply undervoltage: supply +24V',UDINT_TO_DINT(ErrorId),0,0);
		
	16#5180:
		CreateDriveErrMsgDetails := enumMotorEvents.DriveNotEnabled;
		fnLogMsg(ADR(LogMsg_0),LOG_ERROR,'Beckhoff Drive8 ErrorId %d Output stage STO active',UDINT_TO_DINT(ErrorId),0,0);
	16#5181:
		CreateDriveErrMsgDetails := enumMotorEvents.MotorSupplyError;
		fnLogMsg(ADR(LogMsg_0),LOG_ERROR,'Beckhoff Drive8 ErrorId %d Power supply controlword, torque off order',UDINT_TO_DINT(ErrorId),0,0);

	16#5182:
		CreateDriveErrMsgDetails := enumMotorEvents.MotorSupplyError;
		fnLogMsg(ADR(LogMsg_0),LOG_ERROR,'Beckhoff Drive8 ErrorId %d Power supply controlword, live counter inactive',UDINT_TO_DINT(ErrorId),0,0);

	16#5183:
		CreateDriveErrMsgDetails := enumMotorEvents.MotorSupplyError;
		fnLogMsg(ADR(LogMsg_0),LOG_ERROR,'Beckhoff Drive8 ErrorId %d Power supply controlword, NC handling order',UDINT_TO_DINT(ErrorId),0,0);
		
	16#5184:
		CreateDriveErrMsgDetails := enumMotorEvents.MotorSupplyError;
		fnLogMsg(ADR(LogMsg_0),LOG_ERROR,'Beckhoff Drive8 ErrorId %d  Supply DC link circuit is not ready',UDINT_TO_DINT(ErrorId),0,0);
	
	16#5185:
		CreateDriveErrMsgDetails := enumMotorEvents.MotorSupplyError;
		fnLogMsg(ADR(LogMsg_0),LOG_ERROR,'Beckhoff Drive8 ErrorId %d Power supply controlword, non-regenerative brake order',UDINT_TO_DINT(ErrorId),0,0);
	16#5186:
		CreateDriveErrMsgDetails := enumMotorEvents.MotorSupplyError;
		fnLogMsg(ADR(LogMsg_0),LOG_ERROR,'Beckhoff Drive8 ErrorId %d Power supply controlword, regenerative brake order',UDINT_TO_DINT(ErrorId),0,0);
		
	16#5187:
		CreateDriveErrMsgDetails := enumMotorEvents.MotorSupplyError;
		fnLogMsg(ADR(LogMsg_0),LOG_ERROR,'Beckhoff Drive8 ErrorId %d  Power supply communication is not established',UDINT_TO_DINT(ErrorId),0,0);
	16#5190:
		CreateDriveErrMsgDetails := enumMotorEvents.MotorSupplyError;
		fnLogMsg(ADR(LogMsg_0),LOG_ERROR,'Beckhoff Drive8 ErrorId %d  Test 5V supply failed',UDINT_TO_DINT(ErrorId),0,0);

	16#5192:
		CreateDriveErrMsgDetails := enumMotorEvents.MotorSupplyError;
		fnLogMsg(ADR(LogMsg_0),LOG_ERROR,'Beckhoff Drive8 ErrorId %d Supply overvoltage: supply +24V',UDINT_TO_DINT(ErrorId),0,0);

	
	16#5441:
		CreateDriveErrMsgDetails := enumMotorEvents.MotorPositionError;
		fnLogMsg(ADR(LogMsg_0),LOG_ERROR,'Beckhoff Drive8 ErrorId %d  Positive limit switch active',UDINT_TO_DINT(ErrorId),0,0);
	16#5442:
		CreateDriveErrMsgDetails := enumMotorEvents.DriveComError ;
		fnLogMsg(ADR(LogMsg_0),LOG_ERROR,'Beckhoff Drive8 ErrorId %d  Negative limit switch active',UDINT_TO_DINT(ErrorId),0,0);

	16#5580..16#6181:
		CreateDriveErrMsgDetails := enumMotorEvents.MotorGeneralError  ;
		fnLogMsg(ADR(LogMsg_0),LOG_ERROR,'Beckhoff Drive8 ErrorId %d Beckhoff internal Error',UDINT_TO_DINT(ErrorId),0,0);
	16#6182..16#6190:
		CreateDriveErrMsgDetails := enumMotorEvents.MotorGeneralError;
		fnLogMsg(ADR(LogMsg_0),LOG_ERROR,'Beckhoff Drive8 ErrorId %d  Internal Watchdog Error',UDINT_TO_DINT(ErrorId),0,0);
	16#6391..16#639F:
		CreateDriveErrMsgDetails := enumMotorEvents.PLCIllegalParam;
		fnLogMsg(ADR(LogMsg_0),LOG_ERROR,'Beckhoff Drive8 ErrorId %d Operation mode incompatible to PDO',UDINT_TO_DINT(ErrorId),0,0);
	16#63A2..16#63A5:
		CreateDriveErrMsgDetails := enumMotorEvents.MotorFeedBackErr;
		fnLogMsg(ADR(LogMsg_0),LOG_ERROR,'Beckhoff Drive8 ErrorId %d  No position offset',UDINT_TO_DINT(ErrorId),0,0);

	16#63A6..16#63B3:
		CreateDriveErrMsgDetails := enumMotorEvents.PLCIllegalParam ;
		fnLogMsg(ADR(LogMsg_0),LOG_ERROR,'Beckhoff Drive8 ErrorId %d  Jerk factor illegal',UDINT_TO_DINT(ErrorId),0,0);
	
	16#7180:
		CreateDriveErrMsgDetails := enumMotorEvents.MotorSupplyError ;
		fnLogMsg(ADR(LogMsg_0),LOG_ERROR,'Beckhoff Drive8 ErrorId %d Current monitoring error',UDINT_TO_DINT(ErrorId),0,0);


	16#7380:
		CreateDriveErrMsgDetails := enumMotorEvents.MotorSupplyError ;
		fnLogMsg(ADR(LogMsg_0),LOG_ERROR,'Beckhoff Drive8 ErrorId %d Current sensor motor phase U',UDINT_TO_DINT(ErrorId),0,0);
	16#7381:
		CreateDriveErrMsgDetails := enumMotorEvents.MotorSupplyError ;
		fnLogMsg(ADR(LogMsg_0),LOG_ERROR,'Beckhoff Drive8 ErrorId %d  Current sensor motor phase V',UDINT_TO_DINT(ErrorId),0,0);
	16#7382:
		CreateDriveErrMsgDetails := enumMotorEvents.MotorSupplyError ;
		fnLogMsg(ADR(LogMsg_0),LOG_ERROR,'Beckhoff Drive8 ErrorId %d  Current sensor motor phase W',UDINT_TO_DINT(ErrorId),0,0);
	16#8180:
		CreateDriveErrMsgDetails := enumMotorEvents.DriveComError ;
		fnLogMsg(ADR(LogMsg_0),LOG_ERROR,'Beckhoff Drive8 ErrorId %d System restart or sync lost',UDINT_TO_DINT(ErrorId),0,0);
	16#8181:	
		CreateDriveErrMsgDetails := enumMotorEvents.DriveComError ;
		fnLogMsg(ADR(LogMsg_0),LOG_ERROR,'Beckhoff Drive8 ErrorId %d Lost Distributed clocks Sync',UDINT_TO_DINT(ErrorId),0,0);

	16#8185:
		CreateDriveErrMsgDetails := enumMotorEvents.MotorGeneralError ;
		fnLogMsg(ADR(LogMsg_0),LOG_ERROR,'Beckhoff Drive8 ErrorId %d  need an extended fault reset command',UDINT_TO_DINT(ErrorId),0,0);
	16#8611:	
		CreateDriveErrMsgDetails := enumMotorEvents.MotorPositionError ;
		fnLogMsg(ADR(LogMsg_0),LOG_ERROR,'Beckhoff Drive8 ErrorId %d Following error',UDINT_TO_DINT(ErrorId),0,0);

	
	16#8A80..16#8A81:
		CreateDriveErrMsgDetails := enumMotorEvents.PLCIllegalParam ;
		fnLogMsg(ADR(LogMsg_0),LOG_ERROR,'Beckhoff Drive8 ErrorId %d  Illegal Modes Of Operation',UDINT_TO_DINT(ErrorId),0,0);
		
	16#A000..16#A00F :
		CreateDriveErrMsgDetails := enumMotorEvents.MotorGeneralError ;
		fnLogMsg(ADR(LogMsg_0),LOG_ERROR,'Beckhoff Drive8 ErrorId %d  Sync Manager Address Error',UDINT_TO_DINT(ErrorId),0,0);
	
	16#A010..16#A043 :
		CreateDriveErrMsgDetails := enumMotorEvents.PLCIllegalParam ;
		fnLogMsg(ADR(LogMsg_0),LOG_ERROR,'Beckhoff Drive8 ErrorId %d PDO/SDO Error',UDINT_TO_DINT(ErrorId),0,0);
	16#A082:
		CreateDriveErrMsgDetails := enumMotorEvents.MotorGeneralError ;
		fnLogMsg(ADR(LogMsg_0),LOG_ERROR,'Beckhoff Drive8 ErrorId %d  , EtherCAT Slave Stack Error',UDINT_TO_DINT(ErrorId),0,0);
	
	
	16#FF08:
		CreateDriveErrMsgDetails := enumMotorEvents.BreakResistorError ;
		fnLogMsg(ADR(LogMsg_0),LOG_ERROR,'Beckhoff Drive8 ErrorId %d  Shorted Coils Brake',UDINT_TO_DINT(ErrorId),0,0);
	16#FF0C:
		CreateDriveErrMsgDetails := enumMotorEvents.MotorGeneralError ;
		fnLogMsg(ADR(LogMsg_0),LOG_ERROR,'Beckhoff Drive8 ErrorId %d  TorqueOff with emergency brake',UDINT_TO_DINT(ErrorId),0,0);

	16#FFFF:
		CreateDriveErrMsgDetails := enumMotorEvents.MotorGeneralError;
		fnLogMsg(ADR(LogMsg_0),LOG_ERROR,'Beckhoff Drive8 ErrorId %d  Internal Error',UDINT_TO_DINT(ErrorId),0,0);
		
 	ELSE
		fnLogMsg(ADR(LogMsg_0),LOG_ERROR,'unknown Beckhoff Drive8 ErrorId %d ',UDINT_TO_DINT(ErrorId),0,0);
		CreateDriveErrMsgDetails := enumMotorEvents.NoEvents;
END_CASE
END_METHOD

METHOD GetErrCanAdrTemp : BOOL
VAR_INPUT
END_VAR
//Maybe this FB should be remove
CoeErrIdIndex		:= 16#583f;

		
//CoeErrIdIndex	:= 16#603F;
END_METHOD

METHOD Meth_Init : BOOL
VAR_INPUT
END_VAR
ErrorMSgSize := 64;
END_METHOD

END_FUNCTION_BLOCK

// ---- POUs/Lib/Motion/CanOpenAxis/BeckHoff/BeckHoffBasicAxis_FB.TcPOU
FUNCTION_BLOCK PUBLIC BeckHoffBasicAxis_FB EXTENDS CoE_BasicAxis_FB  
VAR_INPUT		
	
END_VAR
VAR_IN_OUT	
END_VAR
VAR_OUTPUT	
END_VAR

VAR
	DebugError					: UINT;
	ErrorMSgSize                : UDINT :=28;
	
END_VAR



SUPER^(AxisRef:=AxisRef);

METHOD CreateDriveErrMsgDetails : enumMotorEvents
VAR_INPUT
	ErrorId			: UDINT;
END_VAR
CASE ErrorId OF
	
	16#1:
		CreateDriveErrMsgDetails := enumMotorEvents.NoEvents;
		fnLogMsg(ADR(LogMsg_0),LOG_ERROR,'BeckHoff Drive ErrorId %d  ,No error',UDINT_TO_DINT(ErrorId),0,0);
	16#4101: 
		CreateDriveErrMsgDetails := enumMotorEvents.MotorOverTemp ;
		fnLogMsg(ADR(LogMsg_0),LOG_ERROR,'BeckHoff Drive ErrorId %d Terminal-Overtemperature',UDINT_TO_DINT(ErrorId),0,0);
	16#4300:
		CreateDriveErrMsgDetails := enumMotorEvents.MotorGeneralError ;
		fnLogMsg(ADR(LogMsg_0),LOG_ERROR,'BeckHoff Drive ErrorId %d Subincrements deactivated',UDINT_TO_DINT(ErrorId),0,0);
	16#4301:
		CreateDriveErrMsgDetails := enumMotorEvents.MotorFeedBackErr ;
		fnLogMsg(ADR(LogMsg_0),LOG_ERROR,'BeckHoff Drive ErrorId %d Encoder-Warning',UDINT_TO_DINT(ErrorId),0,0);
	16#4400:
		CreateDriveErrMsgDetails := enumMotorEvents.MotorGeneralError ;	
		fnLogMsg(ADR(LogMsg_0),LOG_ERROR,'BeckHoff Drive ErrorId %d Drive is not calibrated',UDINT_TO_DINT(ErrorId),0,0);
		
